(* PLC project apollo, CODESYS STW CODESYS V3.5 SP11 - ESX-3CS, author Isoloader *)
(* stored: creationDateTime 2026-05-19T11:25:48.7275673, version 0.1, modificationDateTime 2026-02-02T16:27:17, organization Isoloader *)

TYPE t_pmc_set : ARRAY[1..32] OF t_prog_mov_code;
END_TYPE

TYPE t_prog_mov_diagnostic : (cProgMovDiagnosticDisabled := 0, cProgMovDiagnosticEnabling := 1, cProgMovDiagnosticPrepared := 2, cProgMovDiagnosticActivating := 3, cProgMovDiagnosticWaiting := 4, cProgMovDiagnosticStarting := 5, cProgMovDiagnosticRunning := 6, cProgMovDiagnosticFinishing := 7, cProgMovDiagnosticInterrupted := 8, cProgMovDiagnosticLeaving := 9, cProgMovDiagnosticDeactivatingFromWaiting := 10, cProgMovDiagnosticDeactivatingFromRunning := 11, cProgMovDiagnosticDeactivatingFromFinished := 12, cProgMovDiagnosticDeactivatingFromLeaving := 13, cProgMovDiagnosticInactiveTimeout := 14);
END_TYPE

VAR_GLOBAL  (* GVLallocate *)
  _defaultControllerRotaryEncoderRange : ControllerRotaryEncoderRange;
  _countControllerRotaryEncoderRange : UINT := 0;
  _countControllerMotor : UINT := 0;
END_VAR

VAR_GLOBAL CONSTANT  (* GlobalVariablesApollo *)
  cWinchMotorMaximumVelocityAsHz : REAL := 40.0;
  gSystemApollo : REFERENCE TO SystemApollo;
END_VAR

VAR_GLOBAL CONSTANT  (* GlobalVariablesSpreaderPLC *)
  cRCBrakeSolenoid : USINT := 6;
  cRCBrakePressure : USINT := 7;
  cRCHydraulicFilter : USINT := 8;
  cRCControllerHeartbeat : USINT := 9;
  cRCControllerTempCritical : USINT := 10;
  cRCControllerTempWarning : USINT := 11;
  cRCMotorTempCritical : USINT := 12;
  cRCMotorTempWarning : USINT := 13;
  cRCSideshiftABThrottleError : USINT := 14;
  cRCSideshiftCDThrottleError : USINT := 15;
  cRCPumpThrottleError : USINT := 16;
  cRCAdviseNoFunctionOperatingMode : USINT := 17;
  cRCAdviseSpreaderNotReady : USINT := 18;
  cRCAdviseSpreaderUnableToLockDrive : USINT := 19;
  cRCAdviseNoFunctionUnlessOperational : USINT := 20;
  cRCAdviseTwistlocksNotReady : USINT := 21;
  cRCAdviseNoSideshiftWhenSpreaderLowered : USINT := 22;
END_VAR

FUNCTION allocateControllerMotor : POINTER TO ControllerMotor
  VAR_INPUT
    target : POINTER TO ControllerMotor;
  END_VAR
  VAR
    ptr : POINTER TO ControllerMotor;
  END_VAR

            IF (NOT(target=0)) THEN
	allocateControllerMotor := target;
	RETURN;
END_IF

allocateControllerMotor := __NEW(ControllerMotor);
_countControllerMotor := _countControllerMotor + 1;

IF (allocateControllerMotor=0) THEN
	gCodeErrorHandler(pMessage:='Memory allocation failed for <ControllerMotor>');
END_IF

          
END_FUNCTION

FUNCTION allocateControllerRotaryEncoderRange : REFERENCE TO ControllerRotaryEncoderRange
  VAR_INPUT
    target : REFERENCE TO ControllerRotaryEncoderRange;
  END_VAR
  VAR
    ptr : POINTER TO ControllerRotaryEncoderRange;
  END_VAR

            IF (__ISVALIDREF(target)) THEN
	allocateControllerRotaryEncoderRange REF= target;
	RETURN;
END_IF

ptr := __NEW(ControllerRotaryEncoderRange);
_countControllerRotaryEncoderRange := _countControllerRotaryEncoderRange + 1;

IF (ptr=0) THEN
	gCodeErrorHandler(pMessage:='Memory allocation failed for <ControllerRotaryEncoderRange>');
	allocateControllerRotaryEncoderRange REF= _defaultControllerRotaryEncoderRange;
	RETURN;
END_IF

allocateControllerRotaryEncoderRange REF= ptr^;

          
END_FUNCTION

FUNCTION_BLOCK CANOpenMasterDriveApollo EXTENDS CANOpenMasterDrivePrimary
  VAR
    lWinchAngleA : ControllerRotaryEncoderRange;
    lWinchAngleB : ControllerRotaryEncoderRange;
    lWinchAngleC : ControllerRotaryEncoderRange;
    lWinchAngleD : ControllerRotaryEncoderRange;
    lTransA : ControllerMotor;
    lTransB : ControllerMotor;
    lTransC : ControllerMotor;
    lTransD : ControllerMotor;
    lWinchA : ControllerMotor;
    lWinchB : ControllerMotor;
    lWinchC : ControllerMotor;
    lWinchD : ControllerMotor;
    lSpreader : ControllerSpreader;
  END_VAR

            ;
          

METHOD initialize
                  lTransA.lTypeSteer := FALSE;
lTransB.lTypeSteer := FALSE;
lTransC.lTypeSteer := FALSE;
lTransD.lTypeSteer := FALSE;

lWinchA.lTypeSteer := FALSE;
lWinchB.lTypeSteer := FALSE;
lWinchC.lTypeSteer := FALSE;
lWinchD.lTypeSteer := FALSE;

lWinchAngleA.Name := 'cWinchAngleA';
lWinchAngleA.SubSystem := cSubsystemWinchA;
lWinchAngleA.Sign := -1.0;
lWinchAngleA.UpperObject.Identifier := t_persistent_id.cPersistentID_WinchAUpper;
lWinchAngleA.NetworkId := 2;
registerOperational(ADR(lWinchAngleA));

lWinchAngleB.Name := 'cWinchAngleB';
lWinchAngleB.SubSystem := cSubsystemWinchB;
lWinchAngleB.Sign := 1.0;
lWinchAngleB.UpperObject.Identifier := t_persistent_id.cPersistentID_WinchBUpper;
lWinchAngleB.NetworkId := 2;
registerOperational(ADR(lWinchAngleB));

lWinchAngleC.Name := 'cWinchAngleC';
lWinchAngleC.SubSystem := cSubsystemWinchC;
lWinchAngleC.Sign := -1.0;
lWinchAngleC.UpperObject.Identifier := t_persistent_id.cPersistentID_WinchCUpper;
lWinchAngleC.NetworkId := 2;
registerOperational(ADR(lWinchAngleC));

lWinchAngleD.Name := 'cWinchAngleD';
lWinchAngleD.SubSystem := cSubsystemWinchD;
lWinchAngleD.Sign := 1.0;
lWinchAngleD.UpperObject.Identifier := t_persistent_id.cPersistentID_WinchDUpper;
lWinchAngleD.NetworkId := 2;
registerOperational(ADR(lWinchAngleD));

lTransA.Name := 'cTransA';
lTransA.SubSystem := cSubsystemTravelA;
lTransA.NetworkId := 2;
registerOperational(ADR(lTransA));

lTransB.Name := 'cTransB';
lTransB.SubSystem := cSubsystemTravelB;
lTransB.NetworkId := 2;
registerOperational(ADR(lTransB));

lTransC.Name := 'cTransC';
lTransC.SubSystem := cSubsystemTravelC;
lTransC.NetworkId := 2;
registerOperational(ADR(lTransC));

lTransD.Name := 'cTransD';
lTransD.SubSystem := cSubsystemTravelD;
lTransD.NetworkId := 2;
registerOperational(ADR(lTransD));

lWinchA.Name := 'cWinchA';
lWinchA.SubSystem := cSubsystemWinchA;
lWinchA.NetworkId := 2;	
registerOperational(ADR(lWinchA));

lWinchB.Name := 'cWinchB';
lWinchB.SubSystem := cSubsystemWinchB;
lWinchB.NetworkId := 2;	
registerOperational(ADR(lWinchB));

lWinchC.Name := 'cWinchC';
lWinchC.SubSystem := cSubsystemWinchC;
lWinchC.NetworkId := 2;	
registerOperational(ADR(lWinchC));

lWinchD.Name := 'cWinchD';
lWinchD.SubSystem := cSubsystemWinchD;
lWinchD.NetworkId := 2;	
registerOperational(ADR(lWinchD));

lSpreader.NetworkId := 2;
registerOperational(ADR(lSpreader));

SUPER^.initialize();

lWinchAngleA.lAlarmCANOpenSlaveModulation.registerServer(gSystemApollo.Lift.Interlock);
lWinchAngleB.lAlarmCANOpenSlaveModulation.registerServer(gSystemApollo.Lift.Interlock);
lWinchAngleC.lAlarmCANOpenSlaveModulation.registerServer(gSystemApollo.Lift.Interlock);
lWinchAngleD.lAlarmCANOpenSlaveModulation.registerServer(gSystemApollo.Lift.Interlock);

lWInchA.lAlarmCANOpenSlaveModulation.registerServer(gSystemApollo.Lift.Interlock);
lWInchA.lAlarmCANOpenSlaveBlock.registerServer(gSystemApollo.Lift.Interlock);
lWInchA.lAlarmControllerTemperatureCutback.registerServer(gSystemApollo.Lift.ChargeInterlock);
lWInchA.lAlarmMotorTemperatureCutback.registerServer(gSystemApollo.Lift.ChargeInterlock);
lWInchA.lMaximumVelocity := cWinchMotorMaximumVelocityAsHz;
lWInchA.lAlwaysEnable := TRUE;
lWInchA.lAutomaticEnable := FALSE;

lWInchB.lAlarmCANOpenSlaveModulation.registerServer(gSystemApollo.Lift.Interlock);
lWInchB.lAlarmCANOpenSlaveBlock.registerServer(gSystemApollo.Lift.Interlock);
lWInchB.lAlarmControllerTemperatureCutback.registerServer(gSystemApollo.Lift.ChargeInterlock);
lWInchB.lAlarmMotorTemperatureCutback.registerServer(gSystemApollo.Lift.ChargeInterlock);
lWInchB.lMaximumVelocity := cWinchMotorMaximumVelocityAsHz;
lWInchB.lAlwaysEnable := TRUE;
lWInchB.lAutomaticEnable := FALSE;

lWInchC.lAlarmCANOpenSlaveModulation.registerServer(gSystemApollo.Lift.Interlock);
lWInchC.lAlarmCANOpenSlaveBlock.registerServer(gSystemApollo.Lift.Interlock);
lWInchC.lAlarmControllerTemperatureCutback.registerServer(gSystemApollo.Lift.ChargeInterlock);
lWInchC.lAlarmMotorTemperatureCutback.registerServer(gSystemApollo.Lift.ChargeInterlock);
lWInchC.lMaximumVelocity := cWinchMotorMaximumVelocityAsHz;
lWInchC.lAlwaysEnable := TRUE;
lWInchC.lAutomaticEnable := FALSE;

lWInchD.lAlarmCANOpenSlaveModulation.registerServer(gSystemApollo.Lift.Interlock);
lWInchD.lAlarmCANOpenSlaveBlock.registerServer(gSystemApollo.Lift.Interlock);
lWInchD.lAlarmControllerTemperatureCutback.registerServer(gSystemApollo.Lift.ChargeInterlock);
lWInchD.lAlarmMotorTemperatureCutback.registerServer(gSystemApollo.Lift.ChargeInterlock);
lWInchD.lMaximumVelocity := cWinchMotorMaximumVelocityAsHz;
lWInchD.lAlwaysEnable := TRUE;
lWInchD.lAutomaticEnable := FALSE;

                
END_METHOD

(* {attribute 'monitoring' := 'call'} *)
PROPERTY TransC : REFERENCE TO ControllerMotor
GET
                    TransC REF= lTransC;

                  
END_GET
END_PROPERTY

(* {attribute 'monitoring' := 'call'} *)
PROPERTY WinchD : REFERENCE TO ControllerMotor
GET
                    WinchD REF= lWinchD;

                  
END_GET
END_PROPERTY

(* {attribute 'monitoring' := 'call'} *)
PROPERTY TransD : REFERENCE TO ControllerMotor
GET
                    TransD REF= lTransD;

                  
END_GET
END_PROPERTY

(* {attribute 'monitoring' := 'call'} *)
PROPERTY WinchAngleC : REFERENCE TO ControllerRotaryEncoderRange
GET
                    WinchAngleC REF= lWinchAngleC;

                  
END_GET
END_PROPERTY

(* {attribute 'monitoring' := 'call'} *)
PROPERTY WinchAngleB : REFERENCE TO ControllerRotaryEncoderRange
GET
                    WinchAngleB REF= lWinchAngleB;

                  
END_GET
END_PROPERTY

(* {attribute 'monitoring' := 'call'} *)
PROPERTY TransA : REFERENCE TO ControllerMotor
GET
                    TransA REF= lTransA;

                  
END_GET
END_PROPERTY

(* {attribute 'monitoring' := 'call'} *)
PROPERTY WinchAngleA : REFERENCE TO ControllerRotaryEncoderRange
GET
                    WinchAngleA REF= lWinchAngleA;

                  
END_GET
END_PROPERTY

(* {attribute 'monitoring' := 'call'} *)
PROPERTY WinchC : REFERENCE TO ControllerMotor
GET
                    WinchC REF= lWinchC;

                  
END_GET
END_PROPERTY

(* {attribute 'monitoring' := 'call'} *)
PROPERTY WinchB : REFERENCE TO ControllerMotor
GET
                    WinchB REF= lWinchB;

                  
END_GET
END_PROPERTY

(* {attribute 'monitoring' := 'call'} *)
PROPERTY TransB : REFERENCE TO ControllerMotor
GET
                    TransB REF= lTransB;

                  
END_GET
END_PROPERTY

(* {attribute 'monitoring' := 'call'} *)
PROPERTY WinchAngleD : REFERENCE TO ControllerRotaryEncoderRange
GET
                    WinchAngleD REF= lWinchAngleD;

                  
END_GET
END_PROPERTY

(* {attribute 'monitoring' := 'call'} *)
PROPERTY WinchA : REFERENCE TO ControllerMotor
GET
                    WinchA REF= lWinchA;

                  
END_GET
END_PROPERTY

(* {attribute 'monitoring' := 'call'} *)
PROPERTY Spreader : REFERENCE TO ControllerSpreader
GET
                    Spreader REF= lSpreader;

                  
END_GET
END_PROPERTY
END_FUNCTION_BLOCK

FUNCTION_BLOCK SystemApollo EXTENDS SystemPrimary
  VAR_INPUT
    _CANOpenMasterDriveApollo : REFERENCE TO CANOpenMasterDriveApollo;
    lFunctionalModeControl : FunctionalModeControlApollo;
    lUIEvent : UIEventApollo;
    lProgrammedMovementControl : ProgrammedMovementControl;  (* foobar ProgrammedMovementControlApollo; *)
    lTravel : TravelQuad;
    lLift : LiftQuad;
    lLiftAPositionInterlock : WrapperScaledInterlock;
    lLiftBPositionInterlock : WrapperScaledInterlock;
    lLiftCPositionInterlock : WrapperScaledInterlock;
    lLiftDPositionInterlock : WrapperScaledInterlock;
    lLiftABSynchronousInterlock : SynchronousInterlock;
    lLiftCDSynchronousInterlock : SynchronousInterlock;
    lLiftSynchronousInterlock : SynchronousInterlock;
    lSpreader : Spreader;
    lTwistlockALoweredInterlock : WrapperPositiveOnlyInterlock;
    lTwistlockBLoweredInterlock : WrapperPositiveOnlyInterlock;
    lTwistlockCLoweredInterlock : WrapperPositiveOnlyInterlock;
    lTwistlockDLoweredInterlock : WrapperPositiveOnlyInterlock;
    lTwistlocksReadyInterlock : WrapperTwistlocksReadyInterlock;
    lTwistlockLoweredTravelInterlock : TwistlockLoweredTravelInterlock;
  END_VAR

            ;
          

METHOD initializeStage0
                  IF ((NOT(__ISVALIDREF(gSystemApollo))) OR
	(NOT(__ISVALIDREF(_CANOpenMasterDriveApollo)))) THEN
	gCodeErrorHandler(pMessage:='null reference in SystemApollo');
END_IF

gSystemPrimary REF= gSystemApollo;

_CANOpenMasterDrivePrimary REF= _CANOpenMasterDriveApollo;

_UIEvent REF= lUIEvent;
_FunctionalModeControl REF=  lFunctionalModeControl;
_ProgrammedMovementControl REF= lProgrammedMovementControl;

_Lift REF= lLift;
_Travel REF= lTravel;

SUPER^.initializeStage0();




                
END_METHOD

METHOD initializeStage3
                  registerOperational(ADR(lFunctionalModeControl));
registerOperational(ADR(lUIEvent));
registerOperational(ADR(lProgrammedMovementControl));

registerOperational(ADR(lTravel));
// lTravel.UInterfaceSlowFactor := 0.5; foobar

registerOperational(ADR(lLift));

lLiftAPositionInterlock.Name := 'iLiftAPos';
lLiftAPositionInterlock.Input REF= gSystemApollo.CANOpenMasterDriveApollo.WinchAngleA.PositionObject;
lLiftAPositionInterlock.Client.registerServer(gSystemApollo.Lift.MovementA.Interlock);
lLiftAPositionInterlock.Client.ScalingContext REF= gSystemApollo.Lift.MovementA.InputObject;
lLiftAPositionInterlock.Sign := 1.0;
lLiftAPositionInterlock.SubSystem := cSubsystemWinchA;
registerOperational(ADR(lLiftAPositionInterlock));

lLiftBPositionInterlock.Name := 'iLiftBPos';
lLiftBPositionInterlock.Input REF= gSystemApollo.CANOpenMasterDriveApollo.WinchAngleB.PositionObject;
lLiftBPositionInterlock.Client.registerServer(gSystemApollo.Lift.MovementB.Interlock);
lLiftBPositionInterlock.Client.ScalingContext REF= gSystemApollo.Lift.MovementB.InputObject;
lLiftBPositionInterlock.Sign := 1.0;
lLiftBPositionInterlock.SubSystem := cSubsystemWinchB;
registerOperational(ADR(lLiftBPositionInterlock));

lLiftCPositionInterlock.Name := 'iLiftCPos';
lLiftCPositionInterlock.Input REF= gSystemApollo.CANOpenMasterDriveApollo.WinchAngleC.PositionObject;
lLiftCPositionInterlock.Client.registerServer(gSystemApollo.Lift.MovementC.Interlock);
lLiftCPositionInterlock.Client.ScalingContext REF= gSystemApollo.Lift.MovementC.InputObject;
lLiftCPositionInterlock.Sign := 1.0;
lLiftCPositionInterlock.SubSystem := cSubsystemWinchC;
registerOperational(ADR(lLiftCPositionInterlock));

lLiftDPositionInterlock.Name := 'iLiftDPos';
lLiftDPositionInterlock.Input REF= gSystemApollo.CANOpenMasterDriveApollo.WinchAngleD.PositionObject;
lLiftDPositionInterlock.Client.registerServer(gSystemApollo.Lift.MovementD.Interlock);
lLiftDPositionInterlock.Client.ScalingContext REF= gSystemApollo.Lift.MovementD.InputObject;
lLiftDPositionInterlock.Sign := 1.0;
lLiftDPositionInterlock.SubSystem := cSubsystemWinchD;
registerOperational(ADR(lLiftDPositionInterlock));

lLiftABSynchronousInterlock.Name := 'iLiftABSync';
lLiftABSynchronousInterlock.InputA REF= gSystemApollo.CANOpenMasterDriveApollo.WinchAngleA.PositionObject;
lLiftABSynchronousInterlock.InputB REF= gSystemApollo.CANOpenMasterDriveApollo.WinchAngleB.PositionObject;
lLiftABSynchronousInterlock.ClientA.registerServer(gSystemApollo.Lift.MovementA.Interlock);
lLiftABSynchronousInterlock.ClientA.ScalingContext REF= gSystemApollo.Lift.MovementA.InputObject;
lLiftABSynchronousInterlock.SignA := 1.0;
lLiftABSynchronousInterlock.ClientB.registerServer(gSystemApollo.Lift.MovementB.Interlock);
lLiftABSynchronousInterlock.ClientB.ScalingContext REF= gSystemApollo.Lift.MovementB.InputObject;
lLiftABSynchronousInterlock.SignB := -1.0;
lLiftABSynchronousInterlock.SubSystem := cSubsystemLift;
registerOperational(ADR(lLiftABSynchronousInterlock));

lLiftCDSynchronousInterlock.Name := 'iLiftCDSync';
lLiftCDSynchronousInterlock.InputA REF= gSystemApollo.CANOpenMasterDriveApollo.WinchAngleC.PositionObject;
lLiftCDSynchronousInterlock.InputB REF= gSystemApollo.CANOpenMasterDriveApollo.WinchAngleD.PositionObject;
lLiftCDSynchronousInterlock.ClientA.registerServer(gSystemApollo.Lift.MovementC.Interlock);
lLiftCDSynchronousInterlock.ClientA.ScalingContext REF= gSystemApollo.Lift.MovementC.InputObject;
lLiftCDSynchronousInterlock.SignA := 1.0;
lLiftCDSynchronousInterlock.ClientB.registerServer(gSystemApollo.Lift.MovementD.Interlock);
lLiftCDSynchronousInterlock.ClientB.ScalingContext REF= gSystemApollo.Lift.MovementD.InputObject;
lLiftCDSynchronousInterlock.SignB := -1.0;
lLiftCDSynchronousInterlock.SubSystem := cSubsystemLift;
registerOperational(ADR(lLiftCDSynchronousInterlock));

lLiftSynchronousInterlock.Name := 'iLiftSync';
lLiftSynchronousInterlock.InputA REF= gSystemApollo.lLiftABSynchronousInterlock.AverageObject;
lLiftSynchronousInterlock.InputB REF= gSystemApollo.lLiftCDSynchronousInterlock.AverageObject;
lLiftSynchronousInterlock.ClientA.registerServer(gSystemApollo.Lift.MovementA.Interlock);
lLiftSynchronousInterlock.ClientA.registerServer(gSystemApollo.Lift.MovementB.Interlock);
lLiftSynchronousInterlock.ClientA.ScalingContext REF= gSystemApollo.Lift.InputObject;
lLiftSynchronousInterlock.SignA := 1.0;
lLiftSynchronousInterlock.ClientB.registerServer(gSystemApollo.Lift.MovementC.Interlock);
lLiftSynchronousInterlock.ClientB.registerServer(gSystemApollo.Lift.MovementD.Interlock);
lLiftSynchronousInterlock.ClientB.ScalingContext REF= gSystemApollo.Lift.InputObject;
lLiftSynchronousInterlock.SignB := -1.0;
lLiftSynchronousInterlock.ForceRelaxed := TRUE;
lLiftSynchronousInterlock.SubSystem := cSubsystemLift;
registerOperational(ADR(lLiftSynchronousInterlock));

registerOperational(ADR(lSpreader));

lTwistlockALoweredInterlock.Name := 'iTwistALowered';
lTwistlockALoweredInterlock.Input REF= gSystemApollo.Spreader.TwistlockALoweredStateObject;
lTwistlockALoweredInterlock.Client.registerServer(gSystemApollo.Lift.MovementA.Interlock);
lTwistlockALoweredInterlock.SubSystem := cSubsystemTwistlockA;
registerOperational(ADR(lTwistlockALoweredInterlock));

lTwistlockBLoweredInterlock.Name := 'iTwistBLowered';
lTwistlockBLoweredInterlock.Input REF= gSystemApollo.Spreader.TwistlockBLoweredStateObject;
lTwistlockBLoweredInterlock.Client.registerServer(gSystemApollo.Lift.MovementB.Interlock);
lTwistlockBLoweredInterlock.SubSystem := cSubsystemTwistlockB;
registerOperational(ADR(lTwistlockBLoweredInterlock));

lTwistlockCLoweredInterlock.Name := 'iTwistCLowered';
lTwistlockCLoweredInterlock.Input REF= gSystemApollo.Spreader.TwistlockCLoweredStateObject;
lTwistlockCLoweredInterlock.Client.registerServer(gSystemApollo.Lift.MovementC.Interlock);
lTwistlockCLoweredInterlock.SubSystem := cSubsystemTwistlockC;
registerOperational(ADR(lTwistlockCLoweredInterlock));

lTwistlockDLoweredInterlock.Name := 'iTwistDLowered';
lTwistlockDLoweredInterlock.Input REF= gSystemApollo.Spreader.TwistlockDLoweredStateObject;
lTwistlockDLoweredInterlock.Client.registerServer(gSystemApollo.Lift.MovementD.Interlock);
lTwistlockDLoweredInterlock.SubSystem := cSubsystemTwistlockD;
registerOperational(ADR(lTwistlockDLoweredInterlock));

lTwistlocksReadyInterlock.SubSystem := cSubsystemSpreader;
registerOperational(ADR(lTwistlocksReadyInterlock));

lTwistlockLoweredTravelInterlock.SubSystem := cSubsystemSpreader;
registerOperational(ADR(lTwistlockLoweredTravelInterlock));

SUPER^.initializeStage3();

                
END_METHOD

PROPERTY Spreader : REFERENCE TO Spreader
GET
                    Spreader ref= lSpreader;
                  
END_GET
END_PROPERTY

PROPERTY CANOpenMasterDriveApollo : REFERENCE TO CANOpenMasterDriveApollo
GET
                    CANOpenMasterDriveApollo ref= _CANOpenMasterDriveApollo;
                  
END_GET
END_PROPERTY
END_FUNCTION_BLOCK

FUNCTION_BLOCK ControllerSpreader EXTENDS ControllerSlavePLC
  VAR CONSTANT
    cTelescopingDeadband : t_percentage := 0.05;
    cTransmitPeriod : t_time := TIME#150ms;
    cNominalVoltage : REAL := 120.0;
    cNominalCurrent : REAL := 150.0;
    cPolePairs : REAL := 2.0;
  END_VAR
  VAR
    lPeripheral : PeripheralSpreader;
    lSideshiftABCommand : ValueObjectPercentageOutputReferenceUSINT;
    lSideshiftCDCommand : ValueObjectPercentageOutputReferenceUSINT;
    lTelescopingEnableCommand : ValueObjectBoolOutputReferenceUSINT;
    lTwistlocksLockCommand : ValueObjectBoolOutputReferenceUSINT;
    lTwistlocksUnlockCommand : ValueObjectBoolOutputReferenceUSINT;
    lTelescopingExtendCommand : ValueObjectBoolOutputReferenceUSINT;
    lTelescopingRetractCommand : ValueObjectBoolOutputReferenceUSINT;
    lBrakeDisengageCommand : ValueObjectBoolOutputReferenceUSINT;
    lBrakeThrottleCommand : ValueObjectBoolOutputReferenceUSINT;
    lTelescopingAutoCommand : ValueObjectBoolOutputReferenceUSINT;
    lTelescopingExtendAutoCommand : ValueObjectBool;
    lTelescopingRetractAutoCommand : ValueObjectBool;
    lFaultHydraulicFilter : ValueObjectBoolInputReferenceUINT;
    lBrakeDisengaged : ValueObjectBoolInputReferenceUINT;
    lFaultBrake : ValueObjectBoolInputReferenceUINT;
    lHydraulicPressure : ValueObjectRealScaledOffsetInputReferenceUSINT;
    lHydraulicTemperature : ValueObjectRealScaledOffsetInputReferenceSINT;
    lPumpCurrent : ValueObjectRealScaledOffsetInputReferenceUSINT;
    lPumpBatteryCurrent : ValueObjectRealScaledOffsetInputReferenceUSINT;
    lPumpBatteryVoltage : ValueObjectRealScaledOffsetInputReferenceUINT;
    lPumpVelocity : ValueObjectRealScaledOffsetInputReferenceINT;
    lPumpMotorTemperature : ValueObjectRealScaledOffsetInputReferenceUSINT;
    lPumpControllerTemperature : ValueObjectRealScaledOffsetInputReferenceSINT;
    lPumpState : ValueObjectUSINTInputReferenceUSINT;
    lPumpAllow : ValueObjectBoolInputReferenceUSINT;
    lPumpRunning : ValueObjectBoolInputReferenceUSINT;
    lPumpDirectOn : ValueObjectBoolInputReferenceUSINT;
    lPumpPressureOK : ValueObjectBoolInputReferenceUSINT;
    lPumpAlarm : ValueObjectUINTInputReferenceUINT;
    lTwistlockACurrentState : ValueObjectEnumTypeInputReferenceUINT;
    lTwistlockALoweredState : ValueObjectBoolInputReferenceUINT;
    lTwistlockBCurrentState : ValueObjectEnumTypeInputReferenceUINT;
    lTwistlockBLoweredState : ValueObjectBoolInputReferenceUINT;
    lTwistlockCCurrentState : ValueObjectEnumTypeInputReferenceUINT;
    lTwistlockCLoweredState : ValueObjectBoolInputReferenceUINT;
    lTwistlockDCurrentState : ValueObjectEnumTypeInputReferenceUINT;
    lTwistlockDLoweredState : ValueObjectBoolInputReferenceUINT;
    lTwistlocksCurrentState : ValueObjectEnumTypeInputReferenceUINT;
    lTwistlocksEnabled : ValueObjectBoolInputReferenceUINT;
    lTwistlocksActive : ValueObjectBoolInputReferenceUINT;
    lTelescopingEnabled : ValueObjectBoolInputReferenceUSINT;
    lTelescopingActive : ValueObjectBoolInputReferenceUSINT;
    lTransmitTimer : t_timer;
  END_VAR

            ;
          

METHOD initialize
                  lSideshiftABCommand.initializeValueObjectOp(OpSelf,'SideshiftAB','Sideshift AB command','',cValueStyleConfigurable);
lSideshiftCDCommand.initializeValueObjectOp(OpSelf,'SideshiftCD','Sideshift CD command','',cValueStyleConfigurable);
	
lTelescopingEnableCommand.Index := 0;
lTelescopingEnableCommand.MergeOutput := FALSE;
lTelescopingEnableCommand.initializeValueObjectOp(OpSelf,'TelscpEnbl','Telescoping enabled','',cValueStyleConfigurable);

lTwistlocksLockCommand.Index := 1;
lTwistlocksLockCommand.MergeOutput := TRUE;
lTwistlocksLockCommand.initializeValueObjectOp(OpSelf,'TwstLock','Twistlock lock command','',cValueStyleConfigurable);

lTwistlocksUnlockCommand.Index := 2;
lTwistlocksUnlockCommand.MergeOutput := TRUE;
lTwistlocksUnlockCommand.initializeValueObjectOp(OpSelf,'TwstUnlock','Twistlock unlock command','',cValueStyleConfigurable);

lTelescopingExtendCommand.Index := 3;
lTelescopingExtendCommand.MergeOutput := TRUE;
lTelescopingExtendCommand.initializeValueObjectOp(OpSelf,'TelscpExtend','Telescoping extend command','',cValueStyleConfigurable);

lTelescopingRetractCommand.Index := 4;
lTelescopingRetractCommand.MergeOutput := TRUE;
lTelescopingRetractCommand.initializeValueObjectOp(OpSelf,'TelscpRetract','Telescoping retract command','',cValueStyleConfigurable);

lBrakeDisengageCommand.Index := 5;
lBrakeDisengageCommand.MergeOutput := TRUE;
lBrakeDisengageCommand.initializeValueObjectOp(OpSelf,'BrakeDisengage','Brake disengage command','',cValueStyleConfigurable);

lBrakeThrottleCommand.Index := 6;
lBrakeThrottleCommand.MergeOutput := TRUE;
lBrakeThrottleCommand.initializeValueObjectOp(OpSelf,'BrakeThrottle','Brake throttle','',cValueStyleConfigurable);

lTelescopingAutoCommand.Index := 7;
lTelescopingAutoCommand.MergeOutput := TRUE;
lTelescopingAutoCommand.initializeValueObjectOp(OpSelf,'TelscpAuto','Telescoping auto command enabled','',cValueStyleConfigurable);

lTelescopingExtendAutoCommand.initializeValueObjectOp(OpSelf,'TelscpAutoExt','Telescoping auto extend command','',cValueStyleConfigurable);
lTelescopingRetractAutoCommand.initializeValueObjectOp(OpSelf,'TelscpAutoRet','Telescoping auto retract command','',cValueStyleConfigurable);

lFaultHydraulicFilter.Index := 0;
lFaultHydraulicFilter.initializeValueObjectOp(OpSelf,'HydraulicFilter','Hydraulic filter','',cValueStyleConfigurable);
lBrakeDisengaged.Index := 1;
lBrakeDisengaged.initializeValueObjectOp(OpSelf,'BrakeDisengage','Brake disengage status','',cValueStyleConfigurable);
lFaultBrake.Index := 2;
lFaultBrake.initializeValueObjectOp(OpSelf,'Brake','Brake fault','',cValueStyleConfigurable);
	
lHydraulicPressure.Scaling := 1.0;
lHydraulicPressure.Offset := 0.0;	
lHydraulicPressure.initializeValueObjectOp(OpSelf,'HydPressure','Hydraulic pressure','MPa',cValueStyleConfigurable);

lHydraulicTemperature.Scaling := 1.0;
lHydraulicTemperature.Offset := 0.0;	
lHydraulicTemperature.initializeValueObjectOp(OpSelf,'HydTemp','Hydraulic temperature','celcius',cValueStyleConfigurable);

lPumpCurrent.Scaling := cNominalCurrent/200.0;
lPumpCurrent.initializeValueObjectOp(OpSelf,'PumpCurrent','Hydraulic pump current','amps',cValueStyleConfigurable);

lPumpBatteryCurrent.Scaling := cNominalCurrent/127.0;
lPumpBatteryCurrent.initializeValueObjectOp(OpSelf,'PumpBattCrrnt','Hydraulic pump battery current','amps',cValueStyleConfigurable);

lPumpBatteryVoltage.Scaling := 0.001*cNominalVoltage;
lPumpBatteryVoltage.initializeValueObjectOp(OpSelf,'PumpBattVolt','Hydraulic pump battery voltage','volts',cValueStyleConfigurable);

lPumpVelocity.Scaling := 0.1 / cPolePairs;
lPumpVelocity.initializeValueObjectOp(OpSelf,'PumpVelocity','Hydraulic pump velocity','rpms',cValueStyleConfigurable);

lPumpMotorTemperature.Offset := -40;
lPumpMotorTemperature.initializeValueObjectOp(OpSelf,'PmpMotTemp','Hydraulic pump motor temperature','celcius',cValueStyleConfigurable);

lPumpControllerTemperature.initializeValueObjectOp(OpSelf,'PmpCntrlTemp','Hydraulic pump controller temperature','celcius',cValueStyleConfigurable);

//lPumpState.Index := 0;
lPumpState.initializeValueObjectOp(OpSelf,'PumpState','Hydraulic pump state','rpms',cValueStyleConfigurable);

lPumpAllow.Index := 2;
lPumpAllow.initializeValueObjectOp(OpSelf,'PumpAllow','Hydraulic pump allow status','',cValueStyleConfigurable);

lPumpRunning.Index := 3;
lPumpRunning.initializeValueObjectOp(OpSelf,'PumpRunning','Hydraulic pump running status','',cValueStyleConfigurable);

lPumpDirectOn.Index := 4;
lPumpDirectOn.initializeValueObjectOp(OpSelf,'PumpOn','Hydraulic pump on status','',cValueStyleConfigurable);

lPumpPressureOK.Index := 5;
lPumpPressureOK.initializeValueObjectOp(OpSelf,'PumpPressure','Hydraulic pressure OK status','',cValueStyleConfigurable);

lPumpAlarm.initializeValueObjectOp(OpSelf,'PumpAlarm','Hydraulic pump alarm','',cValueStyleConfigurable);
	
lTwistlockACurrentState.Index := 0;
lTwistlockACurrentState.Length := 2;
lTwistlockACurrentState.EnumType := cEnumTypeLockState;
lTwistlockACurrentState.initializeValueObjectOp(OpSelf,'TwstAStt','Twistlock A state','',cValueStyleConfigurable);

lTwistlockALoweredState.Index := 2;
lTwistlockALoweredState.initializeValueObjectOp(OpSelf,'TwstALow','Twistlock A lowered','',cValueStyleConfigurable);

lTwistlockBCurrentState.Index := 3;
lTwistlockBCurrentState.Length := 2;
lTwistlockBCurrentState.EnumType := cEnumTypeLockState;
lTwistlockBCurrentState.initializeValueObjectOp(OpSelf,'TwstBStt','Twistlock B state','',cValueStyleConfigurable);

lTwistlockBLoweredState.Index := 5;
lTwistlockBLoweredState.initializeValueObjectOp(OpSelf,'TwstBLow','Twistlock B lowered','',cValueStyleConfigurable);

lTwistlockCCurrentState.Index := 6;
lTwistlockCCurrentState.EnumType := cEnumTypeLockState;
lTwistlockCCurrentState.Length := 2;
lTwistlockCCurrentState.initializeValueObjectOp(OpSelf,'TwstCStt','Twistlock C state','',cValueStyleConfigurable);

lTwistlockCLoweredState.Index := 8;
lTwistlockCLoweredState.initializeValueObjectOp(OpSelf,'TwstCLow','Twistlock C lowered','',cValueStyleConfigurable);

lTwistlockDCurrentState.Index := 9;
lTwistlockDCurrentState.EnumType := cEnumTypeLockState;
lTwistlockDCurrentState.Length := 2;
lTwistlockDCurrentState.initializeValueObjectOp(OpSelf,'TwstDStt','Twistlock D state','',cValueStyleConfigurable);

lTwistlockDLoweredState.Index := 11;
lTwistlockDLoweredState.initializeValueObjectOp(OpSelf,'TwstDLow','Twistlock D lowered','',cValueStyleConfigurable);

lTwistlocksCurrentState.Index := 12;
lTwistlocksCurrentState.EnumType := cEnumTypeLockState;
lTwistlocksCurrentState.Length := 2;
lTwistlocksCurrentState.initializeValueObjectOp(OpSelf,'TwstStt','Twistlocks state','',cValueStyleConfigurable);

lTwistlocksEnabled.Index := 14;
lTwistlocksEnabled.initializeValueObjectOp(OpSelf,'TwstEnbl','Twistlocks enabled','',cValueStyleConfigurable);

lTwistlocksActive.Index := 15;
lTwistlocksActive.initializeValueObjectOp(OpSelf,'TwstActive','Twistlocks active','',cValueStyleConfigurable);

lTelescopingEnabled.Index := 0;
lTelescopingEnabled.initializeValueObjectOp(OpSelf,'TelscpEnbl','Telescoping enabled','',cValueStyleConfigurable);
lTelescopingActive.Index := 1;
lTelescopingActive.initializeValueObjectOp(OpSelf,'TelscpActive','Telescoping active','',cValueStyleConfigurable);

SUPER^.initialize();
SubSystem := cSubsystemSpreader;

lPeripheral.initialize();

lAlarmCANOpenSlaveModulation.registerServer(gSystemApollo.Travel.Interlock);
// lAlarmCANOpenSlaveNotOperational.Override := TRUE; //foobar

lStartSystemStateScope := t_system_state.cSystemStateGoOperational;
lOperationalSystemStateScopeLower := t_system_state.cSystemStateOperational;
lModulationSystemStateScope := t_system_state.cSystemStateOperational;

lTransmitTimer.initialize();
lTransmitTimer.Period := cTransmitPeriod;
lTransmitTimer.Enable := TRUE;

// lEnableValidTransmissions := TRUE;
lEnableDetectionTPDO := TRUE;
lEnableNMTDetectionTPDO := TRUE;
lEnableNMTOverrideTPDO := TRUE;
                
END_METHOD

METHOD operator
                  lTwistlocksLockCommand.Value := gSystemApollo.UInterface.TwistlockLock;
lTwistlocksUnlockCommand.Value := gSystemApollo.UInterface.TwistlockUnlock;

lSideshiftABCommand.Value := gSystemApollo.UInterface.SideshiftAB;
lSideshiftCDCommand.Value := gSystemApollo.UInterface.SideshiftCD;

IF (lTelescopingEnabled.Value) THEN
	IF (lTelescopingExtendAutoCommand.Value) THEN
		lTelescopingAutoCommand.Value := TRUE;
		lTelescopingExtendCommand.Value := TRUE;
		lTelescopingRetractCommand.Value := FALSE;
	END_IF

	IF (lTelescopingRetractAutoCommand.Value) THEN
		lTelescopingAutoCommand.Value := TRUE;
		lTelescopingExtendCommand.Value := FALSE;
		lTelescopingRetractCommand.Value := TRUE;
	END_IF
	
	IF (lTelescopingExtendCommand.Value) THEN
		lTelescopingAutoCommand.Value := FALSE;
		lTelescopingExtendCommand.Value := TRUE;
		lTelescopingRetractCommand.Value := FALSE;
	END_IF

	IF (lTelescopingRetractCommand.Value) THEN
		lTelescopingAutoCommand.Value := FALSE;
		lTelescopingExtendCommand.Value := FALSE;
		lTelescopingRetractCommand.Value := TRUE;
	END_IF
ELSE
	lTelescopingAutoCommand.Value := FALSE;
	lTelescopingExtendCommand.Value := FALSE;
	lTelescopingRetractCommand.Value := FALSE;
END_IF

lTransmitTimer.operator();
IF (lTransmitTimer.Expired) THEN
	lTransmitTimer.reset();

	// momentary commands
	lTelescopingEnableCommand.Value := FALSE;
	lTelescopingExtendAutoCommand.Value := FALSE;
	lTelescopingRetractAutoCommand.Value := FALSE;
END_IF

lPeripheral.SupplementaryCommand := 0;

SUPER^.operator();	

lPeripheral.operator();

IF (NOT(ValidTransmissions)) THEN
	// lBrakeDisengaged.Value := FALSE; foobar	
	// RETURN;
END_IF

//foobar error handling

                
END_METHOD

METHOD initializeSpreader
  VAR_INPUT
    supplementaryState : REFERENCE TO UINT;
    hydraulicPressure : REFERENCE TO USINT;
    hydraulicTemperature : REFERENCE TO SINT;
    pumpCurrent : REFERENCE TO USINT;
    pumpBatteryCurrent : REFERENCE TO USINT;
    pumpBatteryVoltage : REFERENCE TO UINT;
    pumpVelocity : REFERENCE TO INT;
    pumpMotorTemperature : REFERENCE TO USINT;
    pumpControllerTemperature : REFERENCE TO SINT;
    pumpState : REFERENCE TO USINT;
    pumpAlarm : REFERENCE TO UINT;
    twistlocksState : REFERENCE TO UINT;
    telescopingState : REFERENCE TO USINT;
    sideshiftABCommand : REFERENCE TO USINT;
    sideshiftCDCommand : REFERENCE TO USINT;
    systemCommand : REFERENCE TO USINT;
  END_VAR
                  lFaultHydraulicFilter.InputReference REF= supplementaryState;
lBrakeDisengaged.InputReference REF= supplementaryState;
lFaultBrake.InputReference REF= supplementaryState;
	
lHydraulicPressure.InputReference REF= hydraulicPressure;
lHydraulicTemperature.InputReference REF= hydraulicTemperature;
lPumpCurrent.InputReference REF= pumpCurrent;
lPumpBatteryCurrent.InputReference REF= pumpBatteryCurrent;
lPumpBatteryVoltage.InputReference ref= pumpBatteryVoltage;
lPumpVelocity.InputReference ref= pumpVelocity;
lPumpMotorTemperature.InputReference ref= pumpMotorTemperature;
lPumpControllerTemperature.InputReference ref= pumpControllerTemperature;
lPumpState.InputReference REF= pumpState;
lPumpAllow.InputReference REF= pumpState;
lPumpRunning.InputReference REF= pumpState;
lPumpDirectOn.InputReference REF= pumpState;
lPumpPressureOK.InputReference REF= pumpState;
lPumpAlarm.InputReference REF= pumpAlarm;
	
lTwistlockACurrentState.InputReference REF= twistlocksState;
lTwistlockALoweredState.InputReference REF= twistlocksState;
lTwistlockBCurrentState.InputReference REF= twistlocksState;
lTwistlockBLoweredState.InputReference REF= twistlocksState;
lTwistlockCCurrentState.InputReference REF= twistlocksState;
lTwistlockCLoweredState.InputReference REF= twistlocksState;
lTwistlockDCurrentState.InputReference REF= twistlocksState;
lTwistlockDLoweredState.InputReference REF= twistlocksState;
lTwistlocksCurrentState.InputReference REF= twistlocksState;

lTwistlocksEnabled.InputReference REF= twistlocksState;
lTwistlocksActive.InputReference REF= twistlocksState;

lTelescopingEnabled.InputReference REF= telescopingState;
lTelescopingActive.InputReference REF= telescopingState;

lSideshiftABCommand.OutputReference REF= sideshiftABCommand;
lSideshiftCDCommand.OutputReference REF= sideshiftCDCommand;

lTelescopingEnableCommand.OutputReference REF= systemCommand;
lTwistlocksLockCommand.OutputReference REF= systemCommand;
lTwistlocksUnlockCommand.OutputReference REF= systemCommand;
lTelescopingExtendCommand.OutputReference REF= systemCommand;
lTelescopingRetractCommand.OutputReference REF= systemCommand;
lBrakeDisengageCommand.OutputReference REF= systemCommand;
lBrakeThrottleCommand.OutputReference REF= systemCommand;
lTelescopingAutoCommand.OutputReference REF= systemCommand;

                
END_METHOD

PROPERTY TwistlockDLoweredState : BOOL
GET
                    TwistlockDLoweredState := lTwistlockDLoweredState.Value;

                  
END_GET
END_PROPERTY

PROPERTY TwistlockDReadyState : BOOL
GET
                    TwistlockDReadyState := ((lTwistlockDCurrentState.Value=t_lock_state.cLockStateLocked) OR
	(lTwistlockDCurrentState.Value=t_lock_state.cLockStateUnlocked));

                  
END_GET
END_PROPERTY

PROPERTY TwistlocksActive : BOOL
GET
                    TwistlocksActive := lTwistlocksActive.Value;

                  
END_GET
END_PROPERTY

PROPERTY TwistlocksCurrentState : t_lock_state
GET
                    TwistlocksCurrentState := lTwistlocksCurrentState.Value;

                  
END_GET
END_PROPERTY

PROPERTY TwistlocksEnabled : BOOL
GET
                    TwistlocksEnabled := lTwistlocksEnabled.Value;

                  
END_GET
END_PROPERTY

PROPERTY TwistlocksLockCommand : BOOL
GET
                    TwistlocksLockCommand := lTwistlocksLockCommand.Value;
                  
END_GET
SET
                    lTwistlocksLockCommand.Value := TwistlocksLockCommand;


                  
END_SET
END_PROPERTY

PROPERTY TwistlocksReadyState : BOOL
GET
                    TwistlocksReadyState := ((lTwistlocksCurrentState.Value=t_lock_state.cLockStateLocked) OR
	(lTwistlocksCurrentState.Value=t_lock_state.cLockStateUnlocked));

                  
END_GET
END_PROPERTY

PROPERTY TwistlocksUnlockCommand : BOOL
GET
                    TwistlocksUnlockCommand := lTwistlocksUnlockCommand.Value;
                  
END_GET
SET
                    lTwistlocksUnlockCommand.Value := TwistlocksUnlockCommand;


                  
END_SET
END_PROPERTY

PROPERTY TypeToken : t_medium_string
GET
                    TypeToken := 'cSpreader';
                  
END_GET
END_PROPERTY

PROPERTY Laden : BOOL
GET
                    Laden := (lTwistlocksCurrentState.Value<>t_lock_state.cLockStateUnlocked);
                  
END_GET
END_PROPERTY

PROPERTY BrakeDisengageCommand : BOOL
GET
                    BrakeDisengageCommand := lBrakeDisengageCommand.Value;
                  
END_GET
SET
                    lBrakeDisengageCommand.Value := BrakeDisengageCommand;

                  
END_SET
END_PROPERTY

PROPERTY BrakeDisengaged : BOOL
GET
                    BrakeDisengaged := lBrakeDisengaged.Value;
                  
END_GET
END_PROPERTY

PROPERTY BrakeThrottleCommand : BOOL
GET
                    BrakeThrottleCommand := lBrakeThrottleCommand.Value;
                  
END_GET
SET
                    lBrakeThrottleCommand.Value := BrakeThrottleCommand;


                  
END_SET
END_PROPERTY

PROPERTY FaultBrake : BOOL
GET
                    FaultBrake := lFaultBrake.Value;
                  
END_GET
END_PROPERTY

PROPERTY FaultHydraulicFilter : BOOL
GET
                    FaultHydraulicFilter := lFaultHydraulicFilter.Value;
                  
END_GET
END_PROPERTY

PROPERTY HydraulicPressure : REAL
GET
                    HydraulicPressure := lHydraulicPressure.Value;

                  
END_GET
END_PROPERTY

PROPERTY HydraulicTemperature : REAL
GET
                    HydraulicTemperature := lHydraulicTemperature.Value;

                  
END_GET
END_PROPERTY

PROPERTY SideshiftABCommand : t_percentage
GET
                    SideshiftABCommand := lSideshiftABCommand.Value;
                  
END_GET
SET
                    lSideshiftABCommand.Value := SideshiftABCommand;


                  
END_SET
END_PROPERTY

PROPERTY SideshiftCDCommand : t_percentage
GET
                    SideshiftCDCommand := lSideshiftCDCommand.Value;
                  
END_GET
SET
                    lSideshiftCDCommand.Value := SideshiftCDCommand;


                  
END_SET
END_PROPERTY

PROPERTY TelescopingActive : BOOL
GET
                    TelescopingActive := lTelescopingActive.Value;

                  
END_GET
END_PROPERTY

PROPERTY TelescopingAutoCommand : BOOL
GET
                    TelescopingAutoCommand := lTelescopingAutoCommand.Value;
                  
END_GET
SET
                    lTelescopingAutoCommand.Value := TelescopingAutoCommand;


                  
END_SET
END_PROPERTY

PROPERTY TelescopingEnableCommand : BOOL
GET
                    TelescopingEnableCommand := lTelescopingEnableCommand.Value;
                  
END_GET
SET
                    lTelescopingEnableCommand.Value := TelescopingEnableCommand;
                  
END_SET
END_PROPERTY

PROPERTY TelescopingEnabled : BOOL
GET
                    TelescopingEnabled := lTelescopingEnabled.Value;

                  
END_GET
END_PROPERTY

PROPERTY TelescopingExtendAutoCommand : BOOL
GET
                    TelescopingExtendAutoCommand := lTelescopingExtendAutoCommand.Value;
                  
END_GET
SET
                    lTelescopingExtendAutoCommand.Value := TelescopingExtendAutoCommand;


                  
END_SET
END_PROPERTY

PROPERTY TelescopingExtendCommand : BOOL
GET
                    TelescopingExtendCommand := lTelescopingExtendCommand.Value;
                  
END_GET
SET
                    lTelescopingExtendCommand.Value := TelescopingExtendCommand;


                  
END_SET
END_PROPERTY

PROPERTY TelescopingRetractAutoCommand : BOOL
GET
                    TelescopingRetractAutoCommand := lTelescopingRetractAutoCommand.Value;
                  
END_GET
SET
                    lTelescopingRetractAutoCommand.Value := TelescopingRetractAutoCommand;


                  
END_SET
END_PROPERTY

PROPERTY TelescopingRetractCommand : BOOL
GET
                    TelescopingRetractCommand := lTelescopingRetractCommand.Value;
                  
END_GET
SET
                    lTelescopingRetractCommand.Value := TelescopingRetractCommand;


                  
END_SET
END_PROPERTY

PROPERTY TwistlockACurrentState : t_lock_state
GET
                    TwistlockACurrentState := lTwistlockACurrentState.Value;

                  
END_GET
END_PROPERTY

PROPERTY TwistlockALoweredState : BOOL
GET
                    TwistlockALoweredState := lTwistlockALoweredState.Value;

                  
END_GET
END_PROPERTY

PROPERTY TwistlockAReadyState : BOOL
GET
                    TwistlockAReadyState := ((lTwistlockACurrentState.Value=t_lock_state.cLockStateLocked) OR
	(lTwistlockACurrentState.Value=t_lock_state.cLockStateUnlocked));

                  
END_GET
END_PROPERTY

PROPERTY TwistlockBCurrentState : t_lock_state
GET
                    TwistlockBCurrentState := lTwistlockBCurrentState.Value;

                  
END_GET
END_PROPERTY

PROPERTY TwistlockBLoweredState : BOOL
GET
                    TwistlockBLoweredState := lTwistlockBLoweredState.Value;

                  
END_GET
END_PROPERTY

PROPERTY TwistlockBReadyState : BOOL
GET
                    TwistlockBReadyState := ((lTwistlockBCurrentState.Value=t_lock_state.cLockStateLocked) OR
	(lTwistlockBCurrentState.Value=t_lock_state.cLockStateUnlocked));

                  
END_GET
END_PROPERTY

PROPERTY TwistlockCCurrentState : t_lock_state
GET
                    TwistlockCCurrentState := lTwistlockCCurrentState.Value;

                  
END_GET
END_PROPERTY

PROPERTY TwistlockCLoweredState : BOOL
GET
                    TwistlockCLoweredState := lTwistlockCLoweredState.Value;

                  
END_GET
END_PROPERTY

PROPERTY TwistlockCReadyState : BOOL
GET
                    TwistlockCReadyState := ((lTwistlockCCurrentState.Value=t_lock_state.cLockStateLocked) OR
	(lTwistlockCCurrentState.Value=t_lock_state.cLockStateUnlocked));

                  
END_GET
END_PROPERTY

PROPERTY TwistlockDCurrentState : t_lock_state
GET
                    TwistlockDCurrentState := lTwistlockDCurrentState.Value;

                  
END_GET
END_PROPERTY

PROPERTY Peripheral : REFERENCE TO Peripheral
GET
                    Peripheral ref= lPeripheral;
                  
END_GET
END_PROPERTY
END_FUNCTION_BLOCK

(* FUNCTION_BLOCK ControllerWinch EXTENDS ControllerMotor400A *)
FUNCTION_BLOCK ControllerWinch EXTENDS ControllerMotor

            ;
          

METHOD initialize
                  SUPER^.initialize();

lAlarmCANOpenSlaveModulation.registerServer(gSystemApollo.Lift.Interlock);
lAlarmCANOpenSlaveBlock.registerServer(gSystemApollo.Lift.Interlock);

lAlarmControllerTemperatureCutback.registerServer(gSystemApollo.Lift.ChargeInterlock);
lAlarmMotorTemperatureCutback.registerServer(gSystemApollo.Lift.ChargeInterlock);

lMaximumVelocity := cWinchMotorMaximumVelocityAsHz;

lAlwaysEnable := TRUE;
lAutomaticEnable := FALSE;

                
END_METHOD
END_FUNCTION_BLOCK

{attribute 'enable_dynamic_creation'}
FUNCTION_BLOCK ControllerWinchAngle EXTENDS ControllerRotaryEncoderRange

            ;
          

METHOD initialize
                  SUPER^.initialize();

lAlarmCANOpenSlaveModulation.registerServer(gSystemApollo.Lift.Interlock);


                
END_METHOD
END_FUNCTION_BLOCK

FUNCTION_BLOCK FunctionalModeControlApollo EXTENDS FunctionalModeControl
  VAR
    lFunctionalModeSpreaderConfiguration : FunctionalModeSpreaderConfiguration;
  END_VAR

            ;
          

METHOD initialize
                  SUPER^.initialize();

lFunctionalModeSpreaderConfiguration.Available := FALSE;
lFunctionalModeSpreaderConfiguration.Enabled := FALSE;
lFunctionalModeSpreaderConfiguration.initialize();

                
END_METHOD

METHOD getMode : REFERENCE TO FunctionalMode
  VAR_INPUT
    mode : t_functional_mode;
  END_VAR
                  getMode REF= lFunctionalModeDefault;
	
CASE mode OF		
	cFunctionalModeDefault:
		getMode REF= lFunctionalModeDefault;	
	cFunctionalModeTravel:
		getMode REF= lFunctionalModeTravel;
	cFunctionalModeLift:
		getMode REF= lFunctionalModeLift;
	cFunctionalModeSpreaderConfiguration:
		getMode REF= lFunctionalModeSpreaderConfiguration;
END_CASE

                
END_METHOD
END_FUNCTION_BLOCK

FUNCTION_BLOCK FunctionalModeSpreaderConfiguration EXTENDS FunctionalMode

            ;
          

METHOD initialize
                  SUPER^.initialize();

lMode := cFunctionalModeSpreaderConfiguration;

                
END_METHOD
END_FUNCTION_BLOCK

FUNCTION_BLOCK LiftAPositionInterlock EXTENDS WrapperScaledInterlock
  VAR CONSTANT
    cOuterRegion : t_percentage := 1.0;
    cInnerRegion : t_percentage := 0.7;
    cInnerValue : t_percentage := 1.0;
    cOuterValue : t_percentage := 0.0;
    cZeroThreshold : t_percentage := 0.03;
  END_VAR

            ;
          

METHOD initialize
                  Name := 'iLiftAPos';

Input REF= gSystemApollo.CANOpenMasterDriveApollo.WinchAngleA.PositionObject;

lTransform.InnerRegion := cInnerRegion;
lTransform.OuterRegion := cOuterRegion;
lTransform.InnerValue := cInnerValue;
lTransform.OuterValue := cOuterValue;

Client.registerServer(gSystemApollo.Lift.MovementA.Interlock);
Client.ScalingContext REF= gSystemApollo.Lift.MovementA.InputObject;
Client.ZeroThreshold := cZeroThreshold;
Sign := 1.0;

SUPER^.initialize();

                
END_METHOD
END_FUNCTION_BLOCK

FUNCTION_BLOCK LiftBPositionInterlock EXTENDS WrapperScaledInterlock
  VAR CONSTANT
    cOuterRegion : t_percentage := 1.0;
    cInnerRegion : t_percentage := 0.7;
    cInnerValue : t_percentage := 1.0;
    cOuterValue : t_percentage := 0.0;
    cZeroThreshold : t_percentage := 0.03;
  END_VAR

            ;
          

METHOD initialize
                  Name := 'iLiftBPos';

Input REF= gSystemApollo.CANOpenMasterDriveApollo.WinchAngleB.PositionObject;

lTransform.InnerRegion := cInnerRegion;
lTransform.OuterRegion := cOuterRegion;
lTransform.InnerValue := cInnerValue;
lTransform.OuterValue := cOuterValue;

Client.registerServer(gSystemApollo.Lift.MovementB.Interlock);
Client.ScalingContext REF= gSystemApollo.Lift.MovementB.InputObject;
Client.ZeroThreshold := cZeroThreshold;
Sign := 1.0;

SUPER^.initialize();

                
END_METHOD
END_FUNCTION_BLOCK

FUNCTION_BLOCK LiftCPositionInterlock EXTENDS WrapperScaledInterlock
  VAR CONSTANT
    cOuterRegion : t_percentage := 1.0;
    cInnerRegion : t_percentage := 0.7;
    cInnerValue : t_percentage := 1.0;
    cOuterValue : t_percentage := 0.0;
    cZeroThreshold : t_percentage := 0.03;
  END_VAR

            ;
          

METHOD initialize
                  Name := 'iLiftCPos';

Input REF= gSystemApollo.CANOpenMasterDriveApollo.WinchAngleC.PositionObject;

lTransform.InnerRegion := cInnerRegion;
lTransform.OuterRegion := cOuterRegion;
lTransform.InnerValue := cInnerValue;
lTransform.OuterValue := cOuterValue;

Client.registerServer(gSystemApollo.Lift.MovementC.Interlock);
Client.ScalingContext REF= gSystemApollo.Lift.MovementC.InputObject;
Client.ZeroThreshold := cZeroThreshold;
Sign := 1.0;

SUPER^.initialize();

                
END_METHOD
END_FUNCTION_BLOCK

FUNCTION_BLOCK LiftDPositionInterlock EXTENDS WrapperScaledInterlock
  VAR CONSTANT
    cOuterRegion : t_percentage := 1.0;
    cInnerRegion : t_percentage := 0.7;
    cInnerValue : t_percentage := 1.0;
    cOuterValue : t_percentage := 0.0;
    cZeroThreshold : t_percentage := 0.03;
  END_VAR

            ;
          

METHOD initialize
                  Name := 'iLiftDPos';

Input REF= gSystemApollo.CANOpenMasterDriveApollo.WinchAngleD.PositionObject;

lTransform.InnerRegion := cInnerRegion;
lTransform.OuterRegion := cOuterRegion;
lTransform.InnerValue := cInnerValue;
lTransform.OuterValue := cOuterValue;

Client.registerServer(gSystemApollo.Lift.MovementD.Interlock);
Client.ScalingContext REF= gSystemApollo.Lift.MovementD.InputObject;
Client.ZeroThreshold := cZeroThreshold;
Sign := 1.0;

SUPER^.initialize();

                
END_METHOD
END_FUNCTION_BLOCK

FUNCTION_BLOCK TwistlockALoweredInterlock EXTENDS WrapperPositiveOnlyInterlock

            ;
          

METHOD initialize
                  Name := 'iTwistALowered';

Input REF= gSystemApollo.Spreader.TwistlockALoweredStateObject;

Client.registerServer(gSystemApollo.Lift.MovementA.Interlock);

SUPER^.initialize();

                
END_METHOD
END_FUNCTION_BLOCK

FUNCTION_BLOCK TwistlockBLoweredInterlock EXTENDS WrapperPositiveOnlyInterlock

            ;
          

METHOD initialize
                  Name := 'iTwistBLowered';

Input REF= gSystemApollo.Spreader.TwistlockBLoweredStateObject;

Client.registerServer(gSystemApollo.Lift.MovementB.Interlock);

SUPER^.initialize();

                
END_METHOD
END_FUNCTION_BLOCK

FUNCTION_BLOCK TwistlockCLoweredInterlock EXTENDS WrapperPositiveOnlyInterlock

            ;
          

METHOD initialize
                  Name := 'iTwistCLowered';

Input REF= gSystemApollo.Spreader.TwistlockCLoweredStateObject;

Client.registerServer(gSystemApollo.Lift.MovementC.Interlock);

SUPER^.initialize();

                
END_METHOD
END_FUNCTION_BLOCK

FUNCTION_BLOCK TwistlockDLoweredInterlock EXTENDS WrapperPositiveOnlyInterlock

            ;
          

METHOD initialize
                  Name := 'iTwistDLowered';

Input REF= gSystemApollo.Spreader.TwistlockDLoweredStateObject;

Client.registerServer(gSystemApollo.Lift.MovementD.Interlock);

SUPER^.initialize();

                
END_METHOD
END_FUNCTION_BLOCK

FUNCTION_BLOCK TwistlockLoweredTravelInterlock EXTENDS WrapperLockoutInterlock

            ;
          

METHOD initialize
                  Name := 'iTwistLowerTrav';

Client.registerServer(gSystemApollo.Travel.Interlock);

SUPER^.initialize();

                
END_METHOD

METHOD operator
                  lInput.Value := ((gSystemApollo.Spreader.TwistlockALoweredState) OR
	(gSystemApollo.Spreader.TwistlockBLoweredState) OR
	(gSystemApollo.Spreader.TwistlockCLoweredState) OR
	(gSystemApollo.Spreader.TwistlockDLoweredState));

SUPER^.operator();

                
END_METHOD
END_FUNCTION_BLOCK

FUNCTION_BLOCK LiftABSynchronousInterlock EXTENDS SynchronousInterlock
  VAR CONSTANT
    cInnerRegion : t_percentage := 0.005;
    cOuterRegion : t_percentage := 0.04;
    cInnerValue : t_percentage := 1.0;
    cOuterValue : t_percentage := 0.0;
    cZeroThreshold : t_percentage := 0.03;
  END_VAR

            
          

METHOD initialize
                  Name := 'iLiftABSync';

InputA REF= gSystemApollo.CANOpenMasterDriveApollo.WinchAngleA.PositionObject;
InputB REF= gSystemApollo.CANOpenMasterDriveApollo.WinchAngleB.PositionObject;

lTransform.InnerRegion := cInnerRegion;
lTransform.OuterRegion := cOuterRegion;
lTransform.InnerValue := cInnerValue;
lTransform.OuterValue := cOuterValue;

ClientA.registerServer(gSystemApollo.Lift.MovementA.Interlock);
ClientA.ScalingContext REF= gSystemApollo.Lift.MovementA.InputObject;
ClientA.ZeroThreshold := cZeroThreshold;
SignA := 1.0;

ClientB.registerServer(gSystemApollo.Lift.MovementB.Interlock);
ClientB.ScalingContext REF= gSystemApollo.Lift.MovementB.InputObject;
ClientB.ZeroThreshold := cZeroThreshold;
SignB := -1.0;

SUPER^.initialize();


                
END_METHOD
END_FUNCTION_BLOCK

FUNCTION_BLOCK LiftCDSynchronousInterlock EXTENDS SynchronousInterlock
  VAR CONSTANT
    cInnerRegion : t_percentage := 0.005;
    cOuterRegion : t_percentage := 0.04;
    cInnerValue : t_percentage := 1.0;
    cOuterValue : t_percentage := 0.0;
    cZeroThreshold : t_percentage := 0.03;
  END_VAR

            ;
          

METHOD initialize
                  Name := 'iLiftCDSync';

InputA REF= gSystemApollo.CANOpenMasterDriveApollo.WinchAngleC.PositionObject;
InputB REF= gSystemApollo.CANOpenMasterDriveApollo.WinchAngleD.PositionObject;

lTransform.InnerRegion := cInnerRegion;
lTransform.OuterRegion := cOuterRegion;
lTransform.InnerValue := cInnerValue;
lTransform.OuterValue := cOuterValue;

ClientA.registerServer(gSystemApollo.Lift.MovementC.Interlock);
ClientA.ScalingContext REF= gSystemApollo.Lift.MovementC.InputObject;
ClientA.ZeroThreshold := cZeroThreshold;
SignA := 1.0;

ClientB.registerServer(gSystemApollo.Lift.MovementD.Interlock);
ClientB.ScalingContext REF= gSystemApollo.Lift.MovementD.InputObject;
ClientB.ZeroThreshold := cZeroThreshold;
SignB := -1.0;

SUPER^.initialize();

                
END_METHOD
END_FUNCTION_BLOCK

FUNCTION_BLOCK LiftSynchronousInterlock EXTENDS SynchronousInterlock
  VAR CONSTANT
    cOuterRegionRelaxed : t_percentage := 0.1;
    cInnerRegionRelaxed : t_percentage := 0.05;
    cInnerValueRelaxed : t_percentage := 1.0;
    cOuterValueRelaxed : t_percentage := 0.0;
    cInnerRegion : t_percentage := 0.005;
    cOuterRegion : t_percentage := 0.04;
    cInnerValue : t_percentage := 1.0;
    cOuterValue : t_percentage := 0.0;
    cZeroThreshold : t_percentage := 0.03;
  END_VAR
  VAR
    lEnableRelaxed : BOOL := FALSE;
  END_VAR

            ;
          

METHOD initialize
                  Name := 'iLiftSync';

InputA REF= gSystemApollo.lLiftABSynchronousInterlock.AverageObject;
InputB REF= gSystemApollo.lLiftCDSynchronousInterlock.AverageObject;

lTransform.InnerRegion := cInnerRegion;
lTransform.OuterRegion := cOuterRegion;
lTransform.InnerValue := cInnerValue;
lTransform.OuterValue := cOuterValue;

ClientA.registerServer(gSystemApollo.Lift.MovementA.Interlock);
ClientA.registerServer(gSystemApollo.Lift.MovementB.Interlock);
ClientA.ScalingContext REF= gSystemApollo.Lift.InputObject;
ClientA.ZeroThreshold := cZeroThreshold;
SignA := 1.0;

ClientB.registerServer(gSystemApollo.Lift.MovementC.Interlock);
ClientB.registerServer(gSystemApollo.Lift.MovementD.Interlock);
ClientB.ScalingContext REF= gSystemApollo.Lift.InputObject;
ClientB.ZeroThreshold := cZeroThreshold;
SignB := -1.0;

SUPER^.initialize();

                
END_METHOD

METHOD operator
                  SUPER^.operator();

IF (lEnableRelaxed) THEN
	lTransform.InnerRegion := cInnerRegionRelaxed;
	lTransform.OuterRegion := cOuterRegionRelaxed;
	lTransform.InnerValue := cInnerValueRelaxed;
	lTransform.OuterValue := cOuterValueRelaxed;
ELSE
	lTransform.InnerRegion := cInnerRegion;
	lTransform.OuterRegion := cOuterRegion;
	lTransform.InnerValue := cInnerValue;
	lTransform.OuterValue := cOuterValue;
END_IF

                
END_METHOD
END_FUNCTION_BLOCK

FUNCTION_BLOCK TwistlocksReadyInterlock EXTENDS ReportableSignedModulation
  VAR
    lPositionLimit : t_percentage := 0.03;  (* machine height dependent *)
    lPosition : t_percentage;
    lResetPosition : t_percentage;
    lAllowAdditionalMovement : BOOL;
  END_VAR

            ;
          

METHOD test
  VAR_INPUT
    override : BOOL;
  END_VAR
                  IF (override) THEN
	RETURN;
END_IF

clear();

lPosition := (gSystemApollo.CANOpenMasterDriveApollo.WinchAngleA.PositionObject.Value +
	gSystemApollo.CANOpenMasterDriveApollo.WinchAngleB.PositionObject.Value +
	gSystemApollo.CANOpenMasterDriveApollo.WinchAngleC.PositionObject.Value +
	gSystemApollo.CANOpenMasterDriveApollo.WinchAngleD.PositionObject.Value) / 4.0;

IF (NOT(gSystemApollo.Spreader.TwistlocksReadyState)) THEN
	lAllowAdditionalMovement := (ABS(lPosition - lResetPosition) < lPositionLimit);

	IF (NOT(lAllowAdditionalMovement)) THEN
		lInterlockState:=cInterlockStateError;
		lScalingPositive := 0.0;
		lThresholdPositive := 0.0;
		lScalingNegative := 0.0;
		lThresholdNegative := 0.0;
		
		trigger(FALSE);
	END_IF
ELSE
	lResetPosition := lPosition;
END_IF

                
END_METHOD

PROPERTY TypeToken : t_medium_string
GET
                    TypeToken := 'iTwistRdy';
                  
END_GET
END_PROPERTY
END_FUNCTION_BLOCK

FUNCTION_BLOCK WrapperTwistlocksReadyInterlock EXTENDS NonOperationalParticleSet
  VAR
    lClient : TwistlocksReadyInterlock;
    lPositionLimit : t_percentage := 0.03;  (* machine height dependent *)
    lPosition : t_percentage;
    lResetPosition : t_percentage;
    lAllowAdditionalMovement : BOOL;
  END_VAR

            ;
          

METHOD initialize
                  Client.initializeState(THIS,'',cCCTwistlocksReadyInterlock);

Client.registerServer(gSystemApollo.Lift.MovementA.Interlock);
Client.registerServer(gSystemApollo.Lift.MovementB.Interlock);
Client.registerServer(gSystemApollo.Lift.MovementC.Interlock);
Client.registerServer(gSystemApollo.Lift.MovementD.Interlock);

SUPER^.initialize();

                
END_METHOD

METHOD operator
                  lClient.test(FALSE);

SUPER^.operator();

                
END_METHOD

PROPERTY Client : REFERENCE TO TwistlocksReadyInterlock
GET
                    Client ref= lClient;
                  
END_GET
END_PROPERTY

PROPERTY TypeToken : t_medium_string
GET
                    TypeToken := 'iwTwistRdy';
                  
END_GET
END_PROPERTY
END_FUNCTION_BLOCK

FUNCTION_BLOCK LiftQuad EXTENDS QuadMovement
  VAR_INPUT
    lEnableBalanceAB : BOOL := FALSE;
  END_VAR
  VAR CONSTANT
    cBalanceABFactor : REAL := 4.0;
    cBalanceADFactor : REAL := 4.0;
    cSlowFactorLaden : t_percentage := 0.6;
    cSlowFactorUnladen : t_percentage := 1.0;
  END_VAR
  VAR
    lBalanceAB : ValueObjectPercentage;
    lBalanceAD : ValueObjectPercentage;
    _ThrottleA : ThrottleMotor;
    _ThrottleB : ThrottleMotor;
    _ThrottleC : ThrottleMotor;
    _ThrottleD : ThrottleMotor;
    lBalanceABFactor : REAL := cBalanceABFactor;
    lBalanceADFactor : REAL := cBalanceADFactor;
    lSlowFactorLaden : t_percentage := cSlowFactorLaden;
    lSlowFactorUnladen : t_percentage := cSlowFactorUnladen;
    lLaden : BOOL := TRUE;
  END_VAR

            ;
          

METHOD checks
                  IF (Laden) THEN
	lFunctionSlowFactor := lSlowFactorLaden;
ELSE
	lFunctionSlowFactor := lSlowFactorUnladen;
END_IF

SUPER^.checks();

                
END_METHOD

METHOD initialize
                  Name := 'Lift';

_ThrottleA.Name := 'ThrottleA';
_ThrottleA.SubSystem := cSubsystemWinchA;
MovementA.SubSystem := cSubsystemWinchA;
MovementA.Throttle REF= _ThrottleA;
_ThrottleA.ControllerMotor REF= gSystemApollo.CANOpenMasterDriveApollo.WinchA;
MovementA.Throttle.Sign := -1.0;
registerNonOperational(ADR(_ThrottleA));

_ThrottleB.Name := 'ThrottleB';
_ThrottleB.SubSystem := cSubsystemWinchB;
MovementB.SubSystem := cSubsystemWinchB;
MovementB.Throttle REF= _ThrottleB;
_ThrottleB.ControllerMotor REF= gSystemApollo.CANOpenMasterDriveApollo.WinchB;
MovementB.Throttle.Sign := 1.0;
registerNonOperational(ADR(_ThrottleB));

_ThrottleC.Name := 'ThrottleC';
_ThrottleC.SubSystem := cSubsystemWinchC;
MovementC.SubSystem := cSubsystemWinchC;
MovementC.Throttle REF= _ThrottleC;
_ThrottleC.ControllerMotor REF= gSystemApollo.CANOpenMasterDriveApollo.WinchC;
MovementC.Throttle.Sign := -1.0;
registerNonOperational(ADR(_ThrottleC));

_ThrottleD.Name := 'ThrottleD';
_ThrottleD.SubSystem := cSubsystemWinchD;
MovementD.SubSystem := cSubsystemWinchD;
MovementD.Throttle REF= _ThrottleD;
_ThrottleD.ControllerMotor REF= gSystemApollo.CANOpenMasterDriveApollo.WinchD;
MovementD.Throttle.Sign := 1.0;
registerNonOperational(ADR(_ThrottleD));

lBalanceAB.Name := 'BalanceAB';
lBalanceAB.SubSystem := cSubsystemLift;
registerNonOperational(ADR(lBalanceAB));

lBalanceAD.Name := 'BalanceAD';
lBalanceAD.SubSystem := cSubsystemLift;
registerNonOperational(ADR(lBalanceAD));

SUPER^.initialize();
SubSystem := cSubsystemLift;

lFunctionalMode := cFunctionalModeLift;

lRegisterUMFSPrimary := TRUE;
lRegisterUMFSAuxilliary := TRUE;
lRegisterUMFSSecondary := TRUE;

lRegisterActive := TRUE;
lRegisterOperatingMode := TRUE;
	
lEnabled := TRUE;
lEnableOnlyOnActiveAllow := FALSE;
lEnableUMFSCheck := TRUE;

lEnableOperatingModeSlow := TRUE;
lEnableUInterfaceSlow := FALSE;
lEnableFunctionSlow := TRUE;

                
END_METHOD

METHOD operator
  VAR
    balanceAB : t_percentage;
    balanceAD : t_percentage;
  END_VAR
                  lInput.InputAsPercentage := gSystemApollo.UInterface.Lift;
lInput.operator();

balanceAB := gSystemApollo.UInterface.LiftBalanceAB;
IF (balanceAB>0) THEN
	balanceAB := MIN(balanceAB * lBalanceABFactor,1.0);
END_IF
IF (balanceAB<0) THEN
	balanceAB := MAX(balanceAB * lBalanceABFactor,-1.0);
END_IF
lBalanceAB.Value := balanceAB;
lBalanceAB.operator();

balanceAD := gSystemApollo.UInterface.LiftBalanceAD;
IF (balanceAD>0) THEN
	balanceAD := MIN(balanceAD * lBalanceADFactor,1.0);
END_IF
IF (balanceAD<0) THEN
	balanceAD := MAX(balanceAD * lBalanceADFactor,-1.0);
END_IF
lBalanceAD.Value := balanceAD;
lBalanceAD.operator();

lScalingA := 1.0;
lScalingB := 1.0;
lScalingC := 1.0;
lScalingD := 1.0;

IF ((lEnableBalanceAB) AND (lBalanceAB.Value<0)) THEN
	lScalingB := lScalingB*ABS(1+lBalanceAB.Value);
	lScalingC := lScalingC*ABS(1+lBalanceAB.Value);
END_IF
IF ((lEnableBalanceAB) AND (lBalanceAB.Value>0)) THEN
	lScalingA := lScalingA*ABS(1-lBalanceAB.Value);
	lScalingD := lScalingD*ABS(1-lBalanceAB.Value);
END_IF

IF (lBalanceAD.Value<0) THEN
	lScalingA := lScalingA*ABS(1+lBalanceAD.Value);
	lScalingB := lScalingB*ABS(1+lBalanceAD.Value);
END_IF
IF (lBalanceAD.Value>0) THEN
	lScalingC := lScalingC*ABS(1-lBalanceAD.Value);
	lScalingD := lScalingD*ABS(1-lBalanceAD.Value);
END_IF

lLaden := gSystemApollo.CANOpenMasterDriveApollo.Spreader.Laden;

SUPER^.operator();

                
END_METHOD

PROPERTY BalanceAB : REFERENCE TO ValueObjectPercentage
GET
                    BalanceAB ref= lBalanceAB;
                  
END_GET
END_PROPERTY

PROPERTY BalanceAD : REFERENCE TO ValueObjectPercentage
GET
                    BalanceAD ref= lBalanceAD;
                  
END_GET
END_PROPERTY

PROPERTY DerivedThrottleA : REFERENCE TO ThrottleMotor
GET
                    DerivedThrottleA ref= _ThrottleA;
                  
END_GET
END_PROPERTY

PROPERTY DerivedThrottleB : REFERENCE TO ThrottleMotor
GET
                    DerivedThrottleB ref= _ThrottleB;
                  
END_GET
END_PROPERTY

PROPERTY DerivedThrottleC : REFERENCE TO ThrottleMotor
GET
                    DerivedThrottleC ref= _ThrottleC;
                  
END_GET
END_PROPERTY

PROPERTY DerivedThrottleD : REFERENCE TO ThrottleMotor
GET
                    DerivedThrottleD ref= _ThrottleD;
                  
END_GET
END_PROPERTY

PROPERTY Laden : BOOL
GET
                    Laden := lLaden;


                  
END_GET
SET
                    lLaden := Laden;
                  
END_SET
END_PROPERTY

PROPERTY TypeToken : t_medium_string
GET
                    TypeToken := 'mLiftQuad';
                  
END_GET
END_PROPERTY
END_FUNCTION_BLOCK

FUNCTION_BLOCK ProgrammedMovementControlApollo EXTENDS ProgrammedMovementControl
  VAR
    lProgMov_Travel_LAT0_Forward : ProgrammedMovementTurn;  (* lProgMov_Lift_Top: ProgrammedMovementLift; lProgMov_Lift_Bottom: ProgrammedMovementLift; lProgMov_Lift_StandardOnGround: ProgrammedMovementLift; lProgMov_Lift_StandardGround: ProgrammedMovementLift; lProgMov_Lift_StandardTruck: ProgrammedMovementLift; lProgMov_Lift_StandardStack1: ProgrammedMovementLift; lProgMov_Lift_StandardStack2: ProgrammedMovementLift; lProgMov_Lift_HicubeOnGround: ProgrammedMovementLift; lProgMov_Lift_HicubeGround: ProgrammedMovementLift; lProgMov_Lift_HicubeTruck: ProgrammedMovementLift; lProgMov_Lift_HicubeStack1: ProgrammedMovementLift; lProgMov_Lift_HicubeStack2: ProgrammedMovementLift; *)
    lProgMov_Travel_LAT0_Reverse : ProgrammedMovementTurn;
    lProgMov_Travel_LAT0_4WS_Forward : ProgrammedMovementTurn;
    lProgMov_Travel_LAT0_4WS_Reverse : ProgrammedMovementTurn;
    lProgMov_Travel_LATPos90_Forward : ProgrammedMovementTurn;
    lProgMov_Travel_LATPos90_Reverse : ProgrammedMovementTurn;
    lProgMov_Travel_LATNeg90_Forward : ProgrammedMovementTurn;
    lProgMov_Travel_LATNeg90_Reverse : ProgrammedMovementTurn;
  END_VAR

            ;
          

METHOD getMovement : REFERENCE TO ProgrammedMovement
  VAR_INPUT
    code : t_prog_mov_code;
  END_VAR
                  getMovement REF= lProgMovNull;

CASE code OF		
		
	(*cProgMovCode_Lift_Top:
		getMovement REF= lProgMov_Lift_Top;	

	cProgMovCode_Lift_Bottom:
		getMovement REF= lProgMov_Lift_Bottom;	
	
	cProgMovCode_Lift_StandardOnGround:
		getMovement REF= lProgMov_Lift_StandardOnGround;	
		
	cProgMovCode_Lift_StandardGround:
		getMovement REF= lProgMov_Lift_StandardGround;	
		
	cProgMovCode_Lift_StandardTruck:
		getMovement REF= lProgMov_Lift_StandardTruck;	

	cProgMovCode_Lift_StandardStack1:
		getMovement REF= lProgMov_Lift_StandardStack1;	
		
	cProgMovCode_Lift_StandardStack2:
		getMovement REF= lProgMov_Lift_StandardStack2;	

	cProgMovCode_Lift_HicubeOnGround:
		getMovement REF= lProgMov_Lift_HicubeOnGround;	
		
	cProgMovCode_Lift_HicubeGround:
		getMovement REF= lProgMov_Lift_HicubeGround;	
		
	cProgMovCode_Lift_HicubeTruck:
		getMovement REF= lProgMov_Lift_HicubeTruck;	

	cProgMovCode_Lift_HicubeStack1:
		getMovement REF= lProgMov_Lift_HicubeStack1;	

	cProgMovCode_Lift_HicubeStack2:
		getMovement REF= lProgMov_Lift_HicubeStack2;*)	
				
	cProgMovCode_Travel_LAT0_Forward:
		getMovement REF= lProgMov_Travel_LAT0_Forward;		

	cProgMovCode_Travel_LAT0_Reverse:
		getMovement REF= lProgMov_Travel_LAT0_Reverse;		

	cProgMovCode_Travel_LAT0_4WS_Forward:
		getMovement REF= lProgMov_Travel_LAT0_4WS_Forward;		

	cProgMovCode_Travel_LAT0_4WS_Reverse:
		getMovement REF= lProgMov_Travel_LAT0_4WS_Reverse;		

	cProgMovCode_Travel_LATPos90_Forward:
		getMovement REF= lProgMov_Travel_LATPos90_Forward;

	cProgMovCode_Travel_LATPos90_Reverse:
		getMovement REF= lProgMov_Travel_LATPos90_Reverse;

	cProgMovCode_Travel_LATNeg90_Forward:
		getMovement REF= lProgMov_Travel_LATNeg90_Forward;

	cProgMovCode_Travel_LATNeg90_Reverse:
		getMovement REF= lProgMov_Travel_LATNeg90_Reverse;

	cProgMovCode_Steer_0:
		getMovement REF= lProgMov_Steer_0;

	cProgMovCode_Test1:
		getMovement REF= lProgMov_Test1;
END_CASE


                
END_METHOD

METHOD getMovementLift : POINTER TO ProgrammedMovementLift
  VAR_INPUT
    code : t_prog_mov_code;
  END_VAR
                  getMovementLift := 0;

CASE code OF
	cProgMovCode_Lift_Top:
		getMovementLift := ADR(lProgMov_Lift_Top);	

	cProgMovCode_Lift_Bottom:
		getMovementLift := ADR(lProgMov_Lift_Bottom);	
	
	cProgMovCode_Lift_StandardOnGround:
		getMovementLift := ADR(lProgMov_Lift_StandardOnGround);	
		
	cProgMovCode_Lift_StandardGround:
		getMovementLift := ADR(lProgMov_Lift_StandardGround);	
		
	cProgMovCode_Lift_StandardTruck:
		getMovementLift := ADR(lProgMov_Lift_StandardTruck);	

	cProgMovCode_Lift_StandardStack1:
		getMovementLift := ADR(lProgMov_Lift_StandardStack1);	
		
	cProgMovCode_Lift_StandardStack2:
		getMovementLift := ADR(lProgMov_Lift_StandardStack2);	

	cProgMovCode_Lift_HicubeOnGround:
		getMovementLift := ADR(lProgMov_Lift_HicubeOnGround);	
		
	cProgMovCode_Lift_HicubeGround:
		getMovementLift := ADR(lProgMov_Lift_HicubeGround);	
		
	cProgMovCode_Lift_HicubeTruck:
		getMovementLift := ADR(lProgMov_Lift_HicubeTruck);	

	cProgMovCode_Lift_HicubeStack1:
		getMovementLift := ADR(lProgMov_Lift_HicubeStack1);	

	cProgMovCode_Lift_HicubeStack2:
		getMovementLift := ADR(lProgMov_Lift_HicubeStack2);
END_CASE


                
END_METHOD

METHOD initialize
                  registerNonOperational(ADR(lProgMovNull));

(*lProgMov_Lift_Top.TargetPositionIdentifier := t_persistent_id.cPersistentID_PMID_Lift_Top;
lProgMov_Lift_Top.Code := cProgMovCode_Lift_Top;
lProgMov_Lift_Top.Name := getStringForProgMovCode(cProgMovCode_Lift_Top);
lProgMov_Lift_Top.PositionZeroThreshold := 0.04;
registerNonOperational(ADR(lProgMov_Lift_Top));

lProgMov_Lift_Bottom.TargetPositionIdentifier := t_persistent_id.cPersistentID_PMID_Lift_Bottom;
lProgMov_Lift_Bottom.Code := cProgMovCode_Lift_Bottom;
lProgMov_Lift_Bottom.Name := getStringForProgMovCode(cProgMovCode_Lift_Bottom);
lProgMov_Lift_Bottom.PositionZeroThreshold := 0.04;
registerNonOperational(ADR(lProgMov_Lift_Bottom));

lProgMov_Lift_StandardOnGround.TargetPositionIdentifier := t_persistent_id.cPersistentID_PMID_Lift_StandardOnGround;
lProgMov_Lift_StandardOnGround.Code := cProgMovCode_Lift_StandardOnGround;
lProgMov_Lift_StandardOnGround.Name := getStringForProgMovCode(cProgMovCode_Lift_StandardOnGround);
lProgMov_Lift_StandardOnGround.PositionZeroThreshold := 0.04;
registerNonOperational(ADR(lProgMov_Lift_StandardOnGround));

lProgMov_Lift_StandardGround.TargetPositionIdentifier := t_persistent_id.cPersistentID_PMID_Lift_StandardGround;
lProgMov_Lift_StandardGround.Code := cProgMovCode_Lift_StandardGround;
lProgMov_Lift_StandardGround.Name := getStringForProgMovCode(cProgMovCode_Lift_StandardGround);
lProgMov_Lift_StandardGround.PositionZeroThreshold := 0.04;
registerNonOperational(ADR(lProgMov_Lift_StandardGround));

lProgMov_Lift_StandardTruck.TargetPositionIdentifier := t_persistent_id.cPersistentID_PMID_Lift_StandardTruck;
lProgMov_Lift_StandardTruck.Code := cProgMovCode_Lift_StandardTruck;
lProgMov_Lift_StandardTruck.Name := getStringForProgMovCode(cProgMovCode_Lift_StandardTruck);
lProgMov_Lift_StandardTruck.PositionZeroThreshold := 0.04;
registerNonOperational(ADR(lProgMov_Lift_StandardTruck));

lProgMov_Lift_StandardStack1.TargetPositionIdentifier := t_persistent_id.cPersistentID_PMID_Lift_StandardStack1;
lProgMov_Lift_StandardStack1.Code := cProgMovCode_Lift_StandardStack1;
lProgMov_Lift_StandardStack1.Name := getStringForProgMovCode(cProgMovCode_Lift_StandardStack1);
lProgMov_Lift_StandardStack1.PositionZeroThreshold := 0.04;
registerNonOperational(ADR(lProgMov_Lift_StandardStack1));

lProgMov_Lift_StandardStack2.TargetPositionIdentifier := t_persistent_id.cPersistentID_PMID_Lift_StandardStack2;
lProgMov_Lift_StandardStack2.Code := cProgMovCode_Lift_StandardStack2;
lProgMov_Lift_StandardStack2.Name := getStringForProgMovCode(cProgMovCode_Lift_StandardStack2);
lProgMov_Lift_StandardStack2.PositionZeroThreshold := 0.04;
registerNonOperational(ADR(lProgMov_Lift_StandardStack2));

lProgMov_Lift_HicubeOnGround.TargetPositionIdentifier := t_persistent_id.cPersistentID_PMID_Lift_HicubeOnGround;
lProgMov_Lift_HicubeOnGround.Code := cProgMovCode_Lift_HicubeOnGround;
lProgMov_Lift_HicubeOnGround.Name := getStringForProgMovCode(cProgMovCode_Lift_HicubeOnGround);
lProgMov_Lift_HicubeOnGround.PositionZeroThreshold := 0.04;
registerNonOperational(ADR(lProgMov_Lift_HicubeOnGround));

lProgMov_Lift_HicubeGround.TargetPositionIdentifier := t_persistent_id.cPersistentID_PMID_Lift_HicubeGround;
lProgMov_Lift_HicubeGround.Code := cProgMovCode_Lift_HicubeGround;
lProgMov_Lift_HicubeGround.Name := getStringForProgMovCode(cProgMovCode_Lift_HicubeGround);
lProgMov_Lift_HicubeGround.PositionZeroThreshold := 0.04;
registerNonOperational(ADR(lProgMov_Lift_HicubeGround));

lProgMov_Lift_HicubeTruck.TargetPositionIdentifier := t_persistent_id.cPersistentID_PMID_Lift_HicubeTruck;
lProgMov_Lift_HicubeTruck.Code := cProgMovCode_Lift_HicubeTruck;
lProgMov_Lift_HicubeTruck.Name := getStringForProgMovCode(cProgMovCode_Lift_HicubeTruck);
lProgMov_Lift_HicubeTruck.PositionZeroThreshold := 0.04;
registerNonOperational(ADR(lProgMov_Lift_HicubeTruck));

lProgMov_Lift_HicubeStack1.TargetPositionIdentifier := t_persistent_id.cPersistentID_PMID_Lift_HicubeStack1;
lProgMov_Lift_HicubeStack1.Code := cProgMovCode_Lift_HicubeStack1;
lProgMov_Lift_HicubeStack1.Name := getStringForProgMovCode(cProgMovCode_Lift_HicubeStack1);
lProgMov_Lift_HicubeStack1.PositionZeroThreshold := 0.04;
registerNonOperational(ADR(lProgMov_Lift_HicubeStack1));

lProgMov_Lift_HicubeStack2.TargetPositionIdentifier := t_persistent_id.cPersistentID_PMID_Lift_HicubeStack2;
lProgMov_Lift_HicubeStack2.Code := cProgMovCode_Lift_HicubeStack2;
lProgMov_Lift_HicubeStack2.Name := getStringForProgMovCode(cProgMovCode_Lift_HicubeStack2);
lProgMov_Lift_HicubeStack2.PositionZeroThreshold := 0.04;
registerNonOperational(ADR(lProgMov_Lift_HicubeStack2));*)

lProgMov_Travel_LAT0_Forward.Code := cProgMovCode_Travel_LAT0_Forward;
lProgMov_Travel_LAT0_Forward.Name := getStringForProgMovCode(cProgMovCode_Travel_LAT0_Forward);
lProgMov_Travel_LAT0_Forward.TargetAngle := 0;
lProgMov_Travel_LAT0_Forward.TargetAngleIncrement := cPi/180.0/3.0;
lProgMov_Travel_LAT0_Forward.TargetAngleZeroThreshold := 0.005;
lProgMov_Travel_LAT0_Forward.TravelThrottle := 0.05;
lProgMov_Travel_LAT0_Forward.SteerModeRequired := cSteerModeLateral;
lProgMov_Travel_LAT0_Forward.SteerModeOnFinishing := cSteerModeLateral;
registerNonOperational(ADR(lProgMov_Travel_LAT0_Forward));

lProgMov_Travel_LAT0_Reverse.Code := cProgMovCode_Travel_LAT0_Reverse;
lProgMov_Travel_LAT0_Reverse.Name := getStringForProgMovCode(cProgMovCode_Travel_LAT0_Reverse);
lProgMov_Travel_LAT0_Reverse.TargetAngle := 0;
lProgMov_Travel_LAT0_Reverse.TargetAngleIncrement := cPi/180.0/3.0;
lProgMov_Travel_LAT0_Reverse.TargetAngleZeroThreshold := 0.005;
lProgMov_Travel_LAT0_Reverse.TravelThrottle := -0.05;
lProgMov_Travel_LAT0_Reverse.SteerModeRequired := cSteerModeLateral;
lProgMov_Travel_LAT0_Reverse.SteerModeOnFinishing := cSteerModeLateral;
registerNonOperational(ADR(lProgMov_Travel_LAT0_Reverse));

lProgMov_Travel_LAT0_4WS_Forward.Code := cProgMovCode_Travel_LAT0_4WS_Forward;
lProgMov_Travel_LAT0_4WS_Forward.Name := getStringForProgMovCode(cProgMovCode_Travel_LAT0_4WS_Forward);
lProgMov_Travel_LAT0_4WS_Forward.TargetAngle := 0;
lProgMov_Travel_LAT0_4WS_Forward.TargetAngleIncrement := cPi/180.0/3.0;
lProgMov_Travel_LAT0_4WS_Forward.TargetAngleZeroThreshold := 0.005;
lProgMov_Travel_LAT0_4WS_Forward.TravelThrottle := 0.05;
lProgMov_Travel_LAT0_4WS_Forward.SteerModeRequired := cSteerModeLateral;
lProgMov_Travel_LAT0_4WS_Forward.SteerModeOnFinishing := cSteerMode4WS;
registerNonOperational(ADR(lProgMov_Travel_LAT0_4WS_Forward));

lProgMov_Travel_LAT0_4WS_Reverse.Code := cProgMovCode_Travel_LAT0_4WS_Reverse;
lProgMov_Travel_LAT0_4WS_Reverse.Name := getStringForProgMovCode(cProgMovCode_Travel_LAT0_4WS_Reverse);
lProgMov_Travel_LAT0_4WS_Reverse.TargetAngle := 0;
lProgMov_Travel_LAT0_4WS_Reverse.TargetAngleIncrement := cPi/180.0/3.0;
lProgMov_Travel_LAT0_4WS_Reverse.TargetAngleZeroThreshold := 0.005;
lProgMov_Travel_LAT0_4WS_Reverse.TravelThrottle := -0.05;
lProgMov_Travel_LAT0_4WS_Reverse.SteerModeRequired := cSteerModeLateral;
lProgMov_Travel_LAT0_4WS_Reverse.SteerModeOnFinishing := cSteerMode4WS;
registerNonOperational(ADR(lProgMov_Travel_LAT0_4WS_Reverse));

lProgMov_Travel_LATPos90_Forward.Code := cProgMovCode_Travel_LATPos90_Forward;
lProgMov_Travel_LATPos90_Forward.Name := getStringForProgMovCode(cProgMovCode_Travel_LATPos90_Forward);
lProgMov_Travel_LATPos90_Forward.TargetAngle := cPiOn2*85.0/90.0;
lProgMov_Travel_LATPos90_Forward.TargetAngleIncrement := cPi/180.0/3.0;
lProgMov_Travel_LATPos90_Forward.TargetAngleZeroThreshold := 0.005;
lProgMov_Travel_LATPos90_Forward.TravelThrottle := 0.05;
lProgMov_Travel_LATPos90_Forward.SteerModeRequired := cSteerModeLateral;
lProgMov_Travel_LATPos90_Forward.SteerModeOnFinishing := cSteerModeLateral;
registerNonOperational(ADR(lProgMov_Travel_LATPos90_Forward));

lProgMov_Travel_LATPos90_Reverse.Code := cProgMovCode_Travel_LATPos90_Reverse;
lProgMov_Travel_LATPos90_Reverse.Name := getStringForProgMovCode(cProgMovCode_Travel_LATPos90_Reverse);
lProgMov_Travel_LATPos90_Reverse.TargetAngle := cPiOn2*85.0/90.0;
lProgMov_Travel_LATPos90_Reverse.TargetAngleIncrement := cPi/180.0/3.0;
lProgMov_Travel_LATPos90_Reverse.TargetAngleZeroThreshold := 0.005;
lProgMov_Travel_LATPos90_Reverse.TravelThrottle := -0.05;
lProgMov_Travel_LATPos90_Reverse.SteerModeRequired := cSteerModeLateral;
lProgMov_Travel_LATPos90_Reverse.SteerModeOnFinishing := cSteerModeLateral;
registerNonOperational(ADR(lProgMov_Travel_LATPos90_Reverse));

lProgMov_Travel_LATNeg90_Forward.Code := cProgMovCode_Travel_LATNeg90_Forward;
lProgMov_Travel_LATNeg90_Forward.Name := getStringForProgMovCode(cProgMovCode_Travel_LATNeg90_Forward);
lProgMov_Travel_LATNeg90_Forward.TargetAngle := -1.0*cPiOn2*85.0/90.0;
lProgMov_Travel_LATNeg90_Forward.TargetAngleIncrement := cPi/180.0/3.0;
lProgMov_Travel_LATNeg90_Forward.TargetAngleZeroThreshold := 0.005;
lProgMov_Travel_LATNeg90_Forward.TravelThrottle := 0.05;
lProgMov_Travel_LATNeg90_Forward.SteerModeRequired := cSteerModeLateral;
lProgMov_Travel_LATNeg90_Forward.SteerModeOnFinishing := cSteerModeLateral;
registerNonOperational(ADR(lProgMov_Travel_LATNeg90_Forward));

lProgMov_Travel_LATNeg90_Reverse.Code := cProgMovCode_Travel_LATNeg90_Reverse;
lProgMov_Travel_LATNeg90_Reverse.Name := getStringForProgMovCode(cProgMovCode_Travel_LATNeg90_Reverse);
lProgMov_Travel_LATNeg90_Reverse.TargetAngle := -1.0*cPiOn2*85.0/90.0;
lProgMov_Travel_LATNeg90_Reverse.TargetAngleIncrement := cPi/180.0/3.0;
lProgMov_Travel_LATNeg90_Reverse.TargetAngleZeroThreshold := 0.005;
lProgMov_Travel_LATNeg90_Reverse.TravelThrottle := -0.05;
lProgMov_Travel_LATNeg90_Reverse.SteerModeRequired := cSteerModeLateral;
lProgMov_Travel_LATNeg90_Reverse.SteerModeOnFinishing := cSteerModeLateral;
registerNonOperational(ADR(lProgMov_Travel_LATNeg90_Reverse));

lProgMov_Steer_0.Code := cProgMovCode_Steer_0;
lProgMov_Steer_0.Name := getStringForProgMovCode(cProgMovCode_Steer_0);
lProgMov_Steer_0.TargetAngle := 0;
lProgMov_Steer_0.TargetAngleIncrement := cPi/180.0/3.0;
lProgMov_Steer_0.TargetAngleZeroThreshold := 0.005;
registerNonOperational(ADR(lProgMov_Steer_0));

lProgMov_Test1.Code := cProgMovCode_Test1;
lProgMov_Test1.Name := getStringForProgMovCode(cProgMovCode_Test1);
lProgMov_Test1.TimeStepMax := 2000;
lProgMov_Test1.registerMovement(cProgMovCode_Travel_LATPos90_Forward);
lProgMov_Test1.registerMovement(cProgMovCode_Travel_LAT0_Forward);
registerNonOperational(ADR(lProgMov_Test1));

lMovement REF= lProgMovNull;

SUPER^.initialize();


                
END_METHOD
END_FUNCTION_BLOCK

FUNCTION_BLOCK ProgrammedMovementLift EXTENDS ProgrammedMovement
  VAR
    lPositionA : REFERENCE TO ValueObjectPercentage;
    lPositionB : REFERENCE TO ValueObjectPercentage;
    lPositionC : REFERENCE TO ValueObjectPercentage;
    lPositionD : REFERENCE TO ValueObjectPercentage;
    lPosition : t_percentage;
    lLiftThrottle : t_percentage := 1.0;
    lTargetPosition : t_persistent_real;
    lTargetThrottleLaden : t_percentage := 0.0;
    lTargetThrottleUnladen : t_percentage := 0.0;
    lAccelerationAsTimeStep : UINT := 20;
    lDecelerationAsPercentage : t_percentage := 0.15;
    lPositionZeroThreshold : REAL := 0.01;
    lSign : REAL := 1.0;
    lPositionAchieved : BOOL;
    lScaling : REAL;
  END_VAR

            ;
          

METHOD disabled
                  SUPER^.disabled();

lPositionAchieved := FALSE;

                
END_METHOD

METHOD initialize
                  SUPER^.initialize();
SubSystem := cSubsystemLift;

lTargetPosition.initialize();

lPositionA REF= gSystemApollo.CANOpenMasterDriveApollo.WinchAngleA.PositionObject;
lPositionB REF= gSystemApollo.CANOpenMasterDriveApollo.WinchAngleB.PositionObject;
lPositionC REF= gSystemApollo.CANOpenMasterDriveApollo.WinchAngleC.PositionObject;
lPositionD REF= gSystemApollo.CANOpenMasterDriveApollo.WinchAngleD.PositionObject;

                
END_METHOD

METHOD running
                  SUPER^.running();

IF (lState<>cProgMovStateRunning) THEN
	RETURN;
END_IF

lScaling := (UINT_TO_REAL(lTimeStep)/UINT_TO_REAL(lAccelerationAsTimeStep));
lScaling := MIN(1.0,lScaling);

lPosition := (lPositionA.Value + lPositionB.Value + lPositionC.Value + lPositionD.Value)/4.0;

lScaling := (lTargetPosition.Value - lPosition)/lDecelerationAsPercentage * lScaling;
lScaling := MIN(1.0,lScaling);
lScaling := MAX(-1.0,lScaling);

IF (ABS(lScaling)<lPositionZeroThreshold) THEN
	lScaling := 0.0;
	lPositionAchieved := TRUE;
END_IF

gSystemApollo.Lift.EnableInputSecondary := TRUE;
gSystemApollo.Lift.InputSecondaryValue := LiftThrottle * lScaling * lSign;

gSystemApollo.lLiftSynchronousInterlock.tighten();

                
END_METHOD

METHOD setPosition
                  lPosition := (lPositionA.Value + lPositionB.Value + lPositionC.Value + lPositionD.Value)/4.0;

TargetPosition := lPosition;
                
END_METHOD

(* {attribute 'monitoring' := 'call'} *)
PROPERTY FinishCondition : BOOL
GET
                    FinishCondition := ((lPositionAchieved) OR
	(lTimeStep>lTimeStepMax));

                  
END_GET
END_PROPERTY

(* {attribute 'monitoring' := 'call'} *)
PROPERTY InterruptCondition : BOOL
GET
                    InterruptCondition := FALSE;

IF (gSystemApollo.UInterface.LiftJoystickInputPresent) THEN
	InterruptCondition := TRUE;	
END_IF
                  
END_GET
END_PROPERTY

PROPERTY LiftThrottle : t_percentage
GET
                    LiftThrottle := lLiftThrottle;
                  
END_GET
SET
                    lLiftThrottle := LiftThrottle;
                  
END_SET
END_PROPERTY

PROPERTY PositionZeroThreshold : REAL
GET
                    PositionZeroThreshold := lPositionZeroThreshold;
                  
END_GET
SET
                    lPositionZeroThreshold := PositionZeroThreshold;
                  
END_SET
END_PROPERTY

(* {attribute 'monitoring' := 'call'} *)
PROPERTY StartCondition : BOOL
GET
                    StartCondition := gSystemApollo.UInterface.AutomationStart;

                  
END_GET
END_PROPERTY

PROPERTY TargetPosition : t_percentage
GET
                    TargetPosition := lTargetPosition.Value;
                  
END_GET
SET
                    lTargetPosition.Value := TargetPosition;
                  
END_SET
END_PROPERTY

PROPERTY TargetPositionIdentifier : t_persistent_id
GET
                    TargetPositionIdentifier := lTargetPosition.Identifier;
                  
END_GET
SET
                    lTargetPosition.Identifier := TargetPositionIdentifier;
                  
END_SET
END_PROPERTY

PROPERTY TypeToken : t_medium_string
GET
                    TypeToken := 'mProgLift';
                  
END_GET
END_PROPERTY
END_FUNCTION_BLOCK

FUNCTION_BLOCK ActiveTravel EXTENDS Active

            ;
          

METHOD transitionOutOfInactive
                  gSystemApollo.CANOpenMasterDriveApollo.TransA.initializeMotorHold();
gSystemApollo.CANOpenMasterDriveApollo.TransB.initializeMotorHold();
gSystemApollo.CANOpenMasterDriveApollo.TransC.initializeMotorHold();
gSystemApollo.CANOpenMasterDriveApollo.TransD.initializeMotorHold();
                
END_METHOD

PROPERTY TypeToken : t_medium_string
GET
                    TypeToken := 'ActiveTravel';
                  
END_GET
END_PROPERTY
END_FUNCTION_BLOCK

FUNCTION_BLOCK TravelDual EXTENDS DualMovement
  VAR CONSTANT
    cSteerStateErrorThrottleThreshold : t_percentage := 0.025;
  END_VAR
  VAR
    lVREnableNullOnSteeringModeChange : ValueReferenceBool;
    lEnableNullOnSteeringModeChange : BOOL := TRUE;
    lVREnableNullOnSteeringState : ValueReferenceBool;
    lEnableNullOnSteeringState : BOOL := TRUE;
    lEnableSteerStateErrorThrottle : BOOL := FALSE;
    _ThrottleA : ThrottleMotor;
    _ThrottleB : ThrottleMotor;
    lSteerStateErrorThrottleThreshold : t_percentage := cSteerStateErrorThrottleThreshold;
  END_VAR

            ;
          

METHOD initialize
                  Name := 'Travel';

lVREnableNullOnSteeringModeChange.initializeValueReference(lEnableNullOnSteeringModeChange,THIS,'NullOnStrModChg');
lVREnableNullOnSteeringState.initializeValueReference(lEnableNullOnSteeringState,THIS,'NullOnStrStt');

_ThrottleA.Name := 'ThrottleA';
MovementA.Throttle REF= _ThrottleA;
_ThrottleA.ControllerMotor REF= gSystemApollo.CANOpenMasterDriveApollo.TransC;
registerNonOperational(ADR(_ThrottleA));

_ThrottleB.Name := 'ThrottleB';
MovementB.Throttle REF= _ThrottleB;
_ThrottleB.ControllerMotor REF= gSystemApollo.CANOpenMasterDriveApollo.TransD;
registerNonOperational(ADR(_ThrottleB));

SUPER^.initialize();

lFunctionalMode := cFunctionalModeDefault;

lRegisterUMFSPrimary := TRUE;
lRegisterUMFSAuxilliary := TRUE;
lRegisterUMFSSecondary := TRUE;

lRegisterActive := TRUE;
lRegisterOperatingMode := TRUE;
	
lEnabled := TRUE;
lEnableOperatingModeSlow := TRUE;
lEnableOnlyOnActiveAllow := FALSE;
lEnableUMFSCheck := TRUE;
                
END_METHOD

METHOD operator
                  lInput.InputAsPercentage := gSystemApollo.UInterface.Travel;
lInput.operator();

IF (lInput.Value<>0) THEN
	lInput.Value := MIN(ABS(lInput.Value),gSystemApollo.Steering.Mode.TravelThrottleThreshold)*lInput.Value/ABS(lInput.Value);
END_IF

IF ((gSystemApollo.Steering.ModeChange) AND 
	(lEnableNullOnSteeringModeChange)) THEN
	lInput.Value := 0;
	//gMessageManager.register(lCode:=cMCAdviseSteerOverideTravelLock);
END_IF

IF ((gSystemApollo.Steering.State=cAdjustStateError) AND 
	(lEnableNullOnSteeringState)) THEN
	IF (lEnableSteerStateErrorThrottle) THEN
		lInput.Value := MIN(ABS(lInput.Value),lSteerStateErrorThrottleThreshold)*lInput.Value/ABS(lInput.Value);
		//gMessageManager.register(lCode:=cMCAdviseSteerOverideTravelLock);
	ELSE
		lInput.Value := 0;
		//gMessageManager.register(lCode:=cMCAdviseSteerOverideTravelLock);		
	END_IF
END_IF

lScalingA := gSystemApollo.Steering.WheelC.WheelVelocityFactor * gSystemApollo.Steering.WheelC.WheelDirection;
lScalingB := gSystemApollo.Steering.WheelD.WheelVelocityFactor * gSystemApollo.Steering.WheelD.WheelDirection;

SUPER^.operator();


                
END_METHOD
END_FUNCTION_BLOCK

FUNCTION_BLOCK TravelQuad EXTENDS QuadMovement
  VAR CONSTANT
    cSteerStateErrorThrottleThreshold : t_percentage := 0.025;
    cSteerAdjustPeriod : t_time := TIME#150ms;
    cBrakePrePeriod : t_time := TIME#500ms;  (* increase from T#200ms to manage brake activation delays *)
    cBrakePostPeriod : t_time := TIME#6s0ms;
    cSlowFactorLaden : t_percentage := 0.6;
    cSlowFactorUnladen : t_percentage := 1.0;
    cFreeWheelOnTurnThreshold : REAL := 0.6;
  END_VAR
  VAR
    lVREnableNullOnSteeringModeChange : ValueReferenceBool;
    lEnableNullOnSteeringModeChange : BOOL := TRUE;
    lVREnableNullOnSteeringState : ValueReferenceBool;
    lEnableNullOnSteeringState : BOOL := TRUE;
    lEnableSteerStateErrorThrottle : BOOL := FALSE;
    lEnableAlwaysActiveOnOperational : BOOL := FALSE;
    lEnableFreeWheelOnTurn : BOOL := FALSE;
    lCausalWaitingForBrakeDisengaged : ReportableCausal;
    _ThrottleA : ThrottleMotor;
    _ThrottleB : ThrottleMotor;
    _ThrottleC : ThrottleMotor;
    _ThrottleD : ThrottleMotor;
    lSteerStateErrorThrottleThreshold : t_percentage := cSteerStateErrorThrottleThreshold;
    lSteerAdjustTimer : t_timer;
    lActiveState : ActiveTravel;
    lSlowFactorLaden : t_percentage := cSlowFactorLaden;
    lSlowFactorUnladen : t_percentage := cSlowFactorUnladen;
  END_VAR

            ;
          

METHOD brake
                  IF (((lInputProcessed<>0) OR
	(lEnableAlwaysActiveOnOperational)) AND
	(gSystemApollo.SystemState.State=cSystemStateOperational)) THEN
	lActiveState.registerActive();
END_IF
lActiveState.operator();

gSystemApollo.CANOpenMasterDriveApollo.Spreader.BrakeDisengageCommand := (lActiveState.IsActive);

// wait until brake has engaged
// evaluating whether to use this mechanism or a timeout on exitOperational, as this state should be protected with a timeout
// deprecated until spreader is reliable in reporting brakeDisengaged status
IF (gSystemApollo.SystemState.State=cSystemStateExitOperational) THEN
	IF (gSystemApollo.CANOpenMasterDriveApollo.Spreader.BrakeDisengaged) THEN
		gSystemApollo.SystemState.transitionAllowDown(cSystemStateExitOperational,ADR(lCausalWaitingForBrakeDisengaged),lCausalWaitingForBrakeDisengaged.Override);
	END_IF
END_IF

// travel case, no explicit holding as stationary
// brake is report as disengaged though no guarantee
// note that input could be zero however
IF ((lActiveState.Allow) AND (gSystemApollo.CANOpenMasterDriveApollo.Spreader.BrakeDisengaged)) THEN
	DerivedThrottleA.ControllerMotor.HoldStationary := FALSE;
	DerivedThrottleB.ControllerMotor.HoldStationary := FALSE;
	DerivedThrottleC.ControllerMotor.HoldStationary := FALSE;
	DerivedThrottleD.ControllerMotor.HoldStationary := FALSE;
	
	RETURN;
END_IF

// pre state or brake may be in unknown state
// force stationary
IF (lActiveState.IsActive) THEN
	DerivedThrottleA.ControllerMotor.HoldStationary := TRUE;
	DerivedThrottleB.ControllerMotor.HoldStationary := TRUE;
	DerivedThrottleC.ControllerMotor.HoldStationary := TRUE;
	DerivedThrottleD.ControllerMotor.HoldStationary := TRUE;
	
	lInputProcessed := 0.0;
	Diagnostic := cMovementDiagnosticBrakeEngaged;

	RETURN;
END_IF

// brake is reported as released, no guarantee that it really is
// can assume that input is zero
// force stationary
// deprecated because keeping the enable bit true does not necessarily force the controller to keep the motor stationary
// it is defined by the aux time parameter in the controller
// assuming that the hold spikes are not being used to keep the controller engaged which is anyway costly in energy
(*IF (gSystemApollo.CANOpenMasterDriveApollo.Spreader.BrakeDisengaged) THEN
	DerivedThrottleA.ControllerMotor.HoldStationary := TRUE;
	DerivedThrottleB.ControllerMotor.HoldStationary := TRUE;
	DerivedThrottleC.ControllerMotor.HoldStationary := TRUE;
	DerivedThrottleD.ControllerMotor.HoldStationary := TRUE;
	
	lInputProcessed := 0.0;
	Diagnostic := cMovementDiagnosticBrakeDisengaged;
	
	RETURN;
END_IF*)

// catchall - clear holding stationary
DerivedThrottleA.ControllerMotor.HoldStationary := FALSE;
DerivedThrottleB.ControllerMotor.HoldStationary := FALSE;
DerivedThrottleC.ControllerMotor.HoldStationary := FALSE;
DerivedThrottleD.ControllerMotor.HoldStationary := FALSE;

                
END_METHOD

METHOD checks
                  IF (lInput.Value<>0) THEN
	IF (gSystemApollo.Steering.Mode.TravelThrottleThreshold=0.0) THEN
		lInputNulled := TRUE;
		Diagnostic := cMovementDiagnosticThreshold;
	END_IF
	InputThresholdAbsolute := ABS(gSystemApollo.Steering.Mode.TravelThrottleThreshold);
END_IF

IF ((gSystemApollo.Steering.ModeChange) AND 
	(lEnableNullOnSteeringModeChange)) THEN
	Diagnostic := cMovementDiagnosticSteeringModeChange;
	lInputNulled := TRUE;
	//gMessageManager.register(lCode:=cMCAdviseSteerOverideTravelLock); //foobar no further notification
END_IF

lSteerAdjustTimer.operator();
IF ((gSystemApollo.Steering.State=cAdjustStateError)
	AND (lEnableNullOnSteeringState)) THEN
	IF (lSteerAdjustTimer.Expired) THEN	
		IF (lEnableSteerStateErrorThrottle) THEN
			lInput.Value := MIN(ABS(lInput.Value),lSteerStateErrorThrottleThreshold)*lInput.Value/ABS(lInput.Value);
		ELSE
			lInputNulled := TRUE;
		END_IF
		
		Diagnostic := cMovementDiagnosticSteeringState;
		//gMessageManager.register(lCode:=cMCAdviseSteerOverideTravelLock); // foobar notification
	END_IF
ELSE
	lSteerAdjustTimer.reset();
END_IF

IF (gSystemApollo.CANOpenMasterDriveApollo.Spreader.Laden) THEN
	lFunctionSlowFactor := lSlowFactorLaden;
ELSE
	lFunctionSlowFactor := lSlowFactorUnladen;
END_IF

SUPER^.checks();

                
END_METHOD

METHOD initialize
                  Name := 'Travel';

lVREnableNullOnSteeringModeChange.initializeValueReference(lEnableNullOnSteeringModeChange,THIS,'NullOnStrModChg','Enable null on steering mode change','',cValueStyleParameter);
lVREnableNullOnSteeringState.initializeValueReference(lEnableNullOnSteeringState,THIS,'NullOnStrStt','Enable null on steering state','',cValueStyleParameter);
	
_ThrottleA.Name := 'ThrottleA';
_ThrottleA.SubSystem := cSubsystemTravelA;
MovementA.SubSystem := cSubsystemTravelA;
MovementA.Throttle REF= _ThrottleA;
_ThrottleA.ControllerMotor REF= gSystemApollo.CANOpenMasterDriveApollo.TransA;
registerNonOperational(ADR(_ThrottleA));

_ThrottleB.Name := 'ThrottleB';
_ThrottleB.SubSystem := cSubsystemTravelB;
MovementB.SubSystem := cSubsystemTravelB;
MovementB.Throttle REF= _ThrottleB;
_ThrottleB.ControllerMotor REF= gSystemApollo.CANOpenMasterDriveApollo.TransB;
registerNonOperational(ADR(_ThrottleB));

_ThrottleC.Name := 'ThrottleC';
_ThrottleC.SubSystem := cSubsystemTravelC;
MovementC.SubSystem := cSubsystemTravelC;
MovementC.Throttle REF= _ThrottleC;
_ThrottleC.ControllerMotor REF= gSystemApollo.CANOpenMasterDriveApollo.TransC;
registerNonOperational(ADR(_ThrottleC));

_ThrottleD.Name := 'ThrottleD';
_ThrottleD.SubSystem := cSubsystemTravelD;
MovementD.SubSystem := cSubsystemTravelD;
MovementD.Throttle REF= _ThrottleD;
_ThrottleD.ControllerMotor REF= gSystemApollo.CANOpenMasterDriveApollo.TransD;
registerNonOperational(ADR(_ThrottleD));

lCausalWaitingForBrakeDisengaged.initializeState(THIS,'',cCCWaitingForBrakeDisengaged);

registerNonOperational(ADR(lActiveState));

SUPER^.initialize();
SubSystem := cSubsystemTravel;

lFunctionalMode := cFunctionalModeDefault;

lRegisterUMFSPrimary := TRUE;
lRegisterUMFSAuxilliary := TRUE;
lRegisterUMFSSecondary := TRUE;

lRegisterActive := TRUE;
lRegisterOperatingMode := TRUE;
	
lEnabled := TRUE;
lEnableOnlyOnActiveAllow := FALSE;
lEnableUMFSCheck := TRUE;

lEnableOperatingModeSlow := TRUE;
lEnableUInterfaceSlow := TRUE;
lEnableFunctionSlow := TRUE;
lEnableBeginnerSlow := TRUE;

lBeginnerSlowFactor := 0.5;
lUInterfaceSlowFactor := 0.5;

lSteerAdjustTimer.initialize();
lSteerAdjustTimer.Enable := TRUE;
lSteerAdjustTimer.Period := cSteerAdjustPeriod;

lActiveState.PrePeriod := cBrakePrePeriod;
lActiveState.PostPeriod := cBrakePostPeriod;

lInterlock.lEnableGradualStop := TRUE;

lInput.Alpha := 1.0;

lEnableAlwaysActiveOnOperational := FALSE;
lEnableFreeWheelOnTurn := TRUE;

gSystemApollo.Steering.WheelA.IndependentWheels := TRUE;
gSystemApollo.Steering.WheelB.IndependentWheels := TRUE;
gSystemApollo.Steering.WheelC.IndependentWheels := TRUE;
gSystemApollo.Steering.WheelD.IndependentWheels := TRUE;

                
END_METHOD

METHOD operator
                  lInput.PreviousAsPercentage := lThrottleValue;
lInput.InputAsPercentage := gSystemApollo.UInterface.Travel;
lInput.operator();

lScalingA := gSystemApollo.Steering.WheelA.WheelVelocityFactor * gSystemApollo.Steering.WheelA.WheelDirection;
lScalingB := gSystemApollo.Steering.WheelB.WheelVelocityFactor * gSystemApollo.Steering.WheelB.WheelDirection;
lScalingC := gSystemApollo.Steering.WheelC.WheelVelocityFactor * gSystemApollo.Steering.WheelC.WheelDirection;
lScalingD := gSystemApollo.Steering.WheelD.WheelVelocityFactor * gSystemApollo.Steering.WheelD.WheelDirection;

IF (lEnableFreeWheelOnTurn) THEN
	_ThrottleA.ControllerMotor.EnableFreeWheel := (ABS(lScalingA)<cFreeWheelOnTurnThreshold);
	_ThrottleB.ControllerMotor.EnableFreeWheel := (ABS(lScalingB)<cFreeWheelOnTurnThreshold);
	_ThrottleC.ControllerMotor.EnableFreeWheel := (ABS(lScalingC)<cFreeWheelOnTurnThreshold);
	_ThrottleD.ControllerMotor.EnableFreeWheel := (ABS(lScalingD)<cFreeWheelOnTurnThreshold);
END_IF

SUPER^.operator();




                
END_METHOD

PROPERTY DerivedThrottleA : REFERENCE TO ThrottleMotor
GET
                    DerivedThrottleA ref= _ThrottleA;
                  
END_GET
END_PROPERTY

PROPERTY DerivedThrottleB : REFERENCE TO ThrottleMotor
GET
                    DerivedThrottleB ref= _ThrottleB;
                  
END_GET
END_PROPERTY

PROPERTY DerivedThrottleC : REFERENCE TO ThrottleMotor
GET
                    DerivedThrottleC ref= _ThrottleC;
                  
END_GET
END_PROPERTY

PROPERTY DerivedThrottleD : REFERENCE TO ThrottleMotor
GET
                    DerivedThrottleD ref= _ThrottleD;
                  
END_GET
END_PROPERTY

PROPERTY TypeToken : t_medium_string
GET
                    TypeToken := 'mTravelQuad';
                  
END_GET
END_PROPERTY
END_FUNCTION_BLOCK

FUNCTION_BLOCK PeripheralSpreader EXTENDS PeripheralPrimary
  VAR
    lAlarmBrakeSolenoid : ReportableAlarm;
    lAlarmBrakePressure : ReportableAlarm;
    lAlarmHydraulicFilter : ReportableAlarm;
    lAlarmControllerHeartbeat : ReportableAlarm;
    lAlarmControllerTempCritical : ReportableAlarm;
    lAlarmControllerTempWarning : ReportableAlarm;
    lAlarmMotorTempCritical : ReportableAlarm;
    lAlarmMotorTempWarning : ReportableAlarm;
    lAlarmSideshiftABThrottleError : ReportableAlarm;
    lAlarmSideshiftCDThrottleError : ReportableAlarm;
    lAlarmPumpThrottleError : ReportableAlarm;
  END_VAR

            ;
          

METHOD initialize
                  //lAlarmSoftware.initializeState(NopSelf,'',cACSoftware);
lAlarmBrakeSolenoid.initializeState(NopSelf,'BrakeSolenoid',cACOutput);
lAlarmBrakePressure.initializeState(NopSelf,'BrakePressure',cACOutput);
lAlarmHydraulicFilter.initializeState(NopSelf,'HydraulicFilter',cACConsumable);

lAlarmControllerHeartbeat.initializeState(NopSelf,'CntHeartbeat',cACHeartbeat);
lAlarmControllerTempCritical.initializeState(NopSelf,'CntTempCrt',cACTemperature);
lAlarmControllerTempWarning.initializeState(NopSelf,'CntTempWrn',cACTemperature);
lAlarmMotorTempCritical.initializeState(NopSelf,'MotTempCrt',cACTemperature);
lAlarmMotorTempWarning.initializeState(NopSelf,'MotTempWrn',cACTemperature);
	
lAlarmSideshiftABThrottleError.initializeState(NopSelf,'SideshiftABThrt',cACOutput);
lAlarmSideshiftCDThrottleError.initializeState(NopSelf,'SideshiftCDThrt',cACOutput);
lAlarmPumpThrottleError.initializeState(NopSelf,'PumpThrt',cACControlSignal);

SUPER^.initialize();

registerReportable(ADR(lAlarmBrakeSolenoid),cRCBrakeSolenoid);
registerReportable(ADR(lAlarmBrakePressure),cRCBrakePressure);
registerReportable(ADR(lAlarmHydraulicFilter),cRCHydraulicFilter);

registerReportable(ADR(lAlarmControllerHeartbeat),cRCControllerHeartbeat);
registerReportable(ADR(lAlarmControllerTempCritical),cRCControllerTempCritical);
registerReportable(ADR(lAlarmControllerTempWarning),cRCControllerTempWarning);
registerReportable(ADR(lAlarmMotorTempCritical),cRCMotorTempCritical);
registerReportable(ADR(lAlarmMotorTempWarning),cRCMotorTempWarning);
	
registerReportable(ADR(lAlarmSideshiftABThrottleError),cRCSideshiftABThrottleError);
registerReportable(ADR(lAlarmSideshiftCDThrottleError),cRCSideshiftCDThrottleError);
registerReportable(ADR(lAlarmPumpThrottleError),cRCPumpThrottleError);

                
END_METHOD
END_FUNCTION_BLOCK

